LIN {X 0,Y 354.946,Z 276.159,A -85,B 0,C 180,E1 -13383.544,E2 -13383.544} C_VEL
LIN {X 0,Y 356.638,Z 285.927,A -85,B 0,C 180,E1 -13386.173,E2 -13386.173} C_VEL
LIN {X 0,Y 356.254,Z 293.138,A -85,B 0,C 180,E1 -13388.006,E2 -13388.006} C_VEL
LIN {X 0,Y 355.986,Z 296.986,A -85,B 0,C 180,E1 -13388.957,E2 -13388.957} C_VEL
LIN {X 0,Y 356.736,Z 302.12,A -85,B 0,C 180,E1 -13389.429,E2 -13389.429} C_VEL
LIN {X 0,Y 360.066,Z 319.74,A -85,B 0,C 180,E1 -13390.451,E2 -13390.451} C_VEL
LIN {X 0,Y 362.277,Z 335.573,A -85,B 0,C 180,E1 -13391.255,E2 -13391.255} C_VEL
LIN {X 0,Y 363.012,Z 348.096,A -85,B 0,C 180,E1 -13391.771,E2 -13391.771} C_VEL
LIN {X 0,Y 361.012,Z 393.9,A -85,B 0,C 180,E1 -13393.203,E2 -13393.203} C_VEL
LIN {X 0,Y 360.015,Z 405.423,A -85,B 0,C 180,E1 -13393.775,E2 -13393.775} C_VEL
LIN {X 0,Y 359.199,Z 414.432,A -85,B 0,C 180,E1 -13394.393,E2 -13394.393} C_VEL
LIN {X 0,Y 358.156,Z 424.02,A -85,B 0,C 180,E1 -13395.221,E2 -13395.221} C_VEL
LIN {X 0,Y 357.004,Z 434.131,A -85,B 0,C 180,E1 -13396.335,E2 -13396.335} C_VEL
LIN {X 0,Y 356.117,Z 442.074,A -85,B 0,C 180,E1 -13397.462,E2 -13397.462} C_VEL
LIN {X 0,Y 355.278,Z 448.663,A -85,B 0,C 180,E1 -13398.59,E2 -13398.59} C_VEL
LIN {X 0,Y 354.683,Z 454.155,A -85,B 0,C 180,E1 -13399.727,E2 -13399.727} C_VEL
LIN {X 0,Y 354.069,Z 459.784,A -85,B 0,C 180,E1 -13401.151,E2 -13401.151} C_VEL
LIN {X 0,Y 353.657,Z 464.249,A -85,B 0,C 180,E1 -13402.578,E2 -13402.578} C_VEL
LIN {X 0,Y 353.348,Z 468.245,A -85,B 0,C 180,E1 -13404.292,E2 -13404.292} C_VEL
LIN {X 0,Y 353.341,Z 470.093,A -85,B 0,C 180,E1 -13405.436,E2 -13405.436} C_VEL
LIN {X 0,Y 353.398,Z 473.622,A -85,B 0,C 180,E1 -13408.86,E2 -13408.86} C_VEL
LIN {X 0,Y 353.4,Z 474.172,A -85,B 0,C 180,E1 -13410,E2 -13410} C_VEL
LIN {X 0,Y 353.339,Z 474.254,A -85,B 0,C 180,E1 -13411.139,E2 -13411.139} C_VEL
LIN {X 0,Y 353.26,Z 473.86,A -85,B 0,C 180,E1 -13412.28,E2 -13412.28} C_VEL
LIN {X 0,Y 353.269,Z 472.879,A -85,B 0,C 180,E1 -13413.421,E2 -13413.421} C_VEL
LIN {X 0,Y 353.323,Z 470.523,A -85,B 0,C 180,E1 -13415.135,E2 -13415.135} C_VEL
LIN {X 0,Y 353.535,Z 466.838,A -85,B 0,C 180,E1 -13416.85,E2 -13416.85} C_VEL
LIN {X 0,Y 353.807,Z 463.697,A -85,B 0,C 180,E1 -13417.993,E2 -13417.993} C_VEL
LIN {X 0,Y 354.266,Z 458.711,A -85,B 0,C 180,E1 -13419.419,E2 -13419.419} C_VEL
LIN {X 0,Y 354.963,Z 452.453,A -85,B 0,C 180,E1 -13420.841,E2 -13420.841} C_VEL
LIN {X 0,Y 355.656,Z 446.355,A -85,B 0,C 180,E1 -13421.975,E2 -13421.975} C_VEL
LIN {X 0,Y 356.361,Z 439.978,A -85,B 0,C 180,E1 -13422.963,E2 -13422.963} C_VEL
LIN {X 0,Y 357.248,Z 432.28,A -85,B 0,C 180,E1 -13423.945,E2 -13423.945} C_VEL
LIN {X 0,Y 358.02,Z 424.21,A -85,B 0,C 180,E1 -13424.785,E2 -13424.785} C_VEL
LIN {X 0,Y 358.803,Z 415.85,A -85,B 0,C 180,E1 -13425.478,E2 -13425.478} C_VEL
LIN {X 0,Y 359.423,Z 407.491,A -85,B 0,C 180,E1 -13426.023,E2 -13426.023} C_VEL
LIN {X 0,Y 360.085,Z 398.162,A -85,B 0,C 180,E1 -13426.469,E2 -13426.469} C_VEL
LIN {X 0,Y 360.556,Z 386.884,A -85,B 0,C 180,E1 -13426.821,E2 -13426.821} C_VEL
LIN {X 0,Y 361.133,Z 345.094,A -85,B 0,C 180,E1 -13427.675,E2 -13427.675} C_VEL
LIN {X 0,Y 358.638,Z 327.17,A -85,B 0,C 180,E1 -13428.215,E2 -13428.215} C_VEL
LIN {X 0,Y 355.966,Z 312.815,A -85,B 0,C 180,E1 -13428.71,E2 -13428.71} C_VEL
LIN {X 0,Y 357.346,Z 297.3,A -85,B 0,C 180,E1 -13432.676,E2 -13432.676} C_VEL
LIN {X 0,Y 357.807,Z 292.005,A -85,B 0,C 180,E1 -13434.052,E2 -13434.052} C_VEL
LIN {X 0,Y 356.54,Z 283.93,A -85,B 0,C 180,E1 -13436.328,E2 -13436.328} C_VEL
LIN {X 0,Y 354.88,Z 276.094,A -85,B 0,C 180,E1 -13438.684,E2 -13438.684} C_VEL
LIN {X 0,Y 354.795,Z 276.096,A -85,B 0,C 180,E1 -13442.332,E2 -13442.332} C_VEL
LIN {X 0,Y 354.827,Z 276.09,A -85,B 0,C 180,E1 -13445.697,E2 -13445.697} C_VEL
LIN {X 0,Y 354.808,Z 276.101,A -85,B 0,C 180,E1 -13449.417,E2 -13449.417} C_VEL
LIN {X 0,Y 354.796,Z 276.102,A -85,B 0,C 180,E1 -13452.865,E2 -13452.865} C_VEL
LIN {X 0,Y 354.775,Z 276.104,A -85,B 0,C 180,E1 -13456.102,E2 -13456.102} C_VEL
LIN {X 0,Y 354.774,Z 276.105,A -85,B 0,C 180,E1 -13459.174,E2 -13459.174} C_VEL
LIN {X 0,Y 354.808,Z 276.099,A -85,B 0,C 180,E1 -13462.402,E2 -13462.402} C_VEL
LIN {X 0,Y 354.819,Z 276.092,A -85,B 0,C 180,E1 -13464.939,E2 -13464.939} C_VEL
LIN {X 0,Y 354.8,Z 276.094,A -85,B 0,C 180,E1 -13468.403,E2 -13468.403} C_VEL
LIN {X 0,Y 354.81,Z 276.103,A -85,B 0,C 180,E1 -13471.612,E2 -13471.612} C_VEL
LIN {X 0,Y 354.858,Z 276.093,A -85,B 0,C 180,E1 -13475.421,E2 -13475.421} C_VEL
LIN {X 0,Y 354.833,Z 276.087,A -85,B 0,C 180,E1 -13479.11,E2 -13479.11} C_VEL
LIN {X 0,Y 354.885,Z 276.084,A -85,B 0,C 180,E1 -13482.716,E2 -13482.716} C_VEL
LIN {X 0,Y 354.956,Z 276.08,A -85,B 0,C 180,E1 -13486.252,E2 -13486.252} C_VEL
LIN {X 0,Y 354.981,Z 276.068,A -85,B 0,C 180,E1 -13489.733,E2 -13489.733} C_VEL
LIN {X 0,Y 355.127,Z 276.053,A -85,B 0,C 180,E1 -13493.177,E2 -13493.177} C_VEL
LIN {X 0,Y 355.234,Z 276.044,A -85,B 0,C 180,E1 -13497.729,E2 -13497.729} C_VEL
LIN {X 0,Y 355.352,Z 276.022,A -85,B 0,C 180,E1 -13499.996,E2 -13499.996} C_VEL
LIN {X 0,Y 355.24,Z 276.047,A -85,B 0,C 180,E1 -13502.264,E2 -13502.264} C_VEL
LIN {X 0,Y 355.096,Z 276.061,A -85,B 0,C 180,E1 -13506.816,E2 -13506.816} C_VEL
LIN {X 0,Y 354.951,Z 276.076,A -85,B 0,C 180,E1 -13510.261,E2 -13510.261} C_VEL
LIN {X 0,Y 354.937,Z 276.086,A -85,B 0,C 180,E1 -13514.015,E2 -13514.015} C_VEL
LIN {X 0,Y 354.914,Z 276.088,A -85,B 0,C 180,E1 -13518.104,E2 -13518.104} C_VEL
LIN {X 0,Y 354.824,Z 276.098,A -85,B 0,C 180,E1 -13522.102,E2 -13522.102} C_VEL
LIN {X 0,Y 354.887,Z 276.088,A -85,B 0,C 180,E1 -13525.823,E2 -13525.823} C_VEL
LIN {X 0,Y 354.803,Z 276.1,A -85,B 0,C 180,E1 -13529.678,E2 -13529.678} C_VEL
LIN {X 0,Y 354.789,Z 276.102,A -85,B 0,C 180,E1 -13533.698,E2 -13533.698} C_VEL
LIN {X 0,Y 354.779,Z 276.093,A -85,B 0,C 180,E1 -13536.456,E2 -13536.456} C_VEL
LIN {X 0,Y 354.804,Z 276.097,A -85,B 0,C 180,E1 -13539.42,E2 -13539.42} C_VEL
LIN {X 0,Y 354.819,Z 276.1,A -85,B 0,C 180,E1 -13542.873,E2 -13542.873} C_VEL
LIN {X 0,Y 354.844,Z 276.098,A -85,B 0,C 180,E1 -13546.116,E2 -13546.116} C_VEL
LIN {X 0,Y 354.831,Z 276.097,A -85,B 0,C 180,E1 -13549.185,E2 -13549.185} C_VEL
LIN {X 0,Y 354.844,Z 276.163,A -85,B 0,C 180,E1 -13552.213,E2 -13552.213} C_VEL
LIN {X 0,Y 356.19,Z 282.921,A -85,B 0,C 180,E1 -13554.336,E2 -13554.336} C_VEL
LIN {X 0,Y 359.045,Z 291.373,A -85,B 0,C 180,E1 -13554.722,E2 -13554.722} C_VEL
LIN {X 0,Y 361.86,Z 303.963,A -85,B 0,C 180,E1 -13555.175,E2 -13555.175} C_VEL
LIN {X 0,Y 360.834,Z 359.468,A -85,B 0,C 180,E1 -13556.325,E2 -13556.325} C_VEL
LIN {X 0,Y 360.551,Z 369.013,A -85,B 0,C 180,E1 -13556.672,E2 -13556.672} C_VEL
LIN {X 0,Y 360.038,Z 379.383,A -85,B 0,C 180,E1 -13557.226,E2 -13557.226} C_VEL
LIN {X 0,Y 359.213,Z 390.94,A -85,B 0,C 180,E1 -13558.113,E2 -13558.113} C_VEL
LIN {X 0,Y 358.442,Z 399.876,A -85,B 0,C 180,E1 -13559.024,E2 -13559.024} C_VEL
LIN {X 0,Y 357.714,Z 407.018,A -85,B 0,C 180,E1 -13559.919,E2 -13559.919} C_VEL
LIN {X 0,Y 356.986,Z 413.17,A -85,B 0,C 180,E1 -13560.84,E2 -13560.84} C_VEL
LIN {X 0,Y 356.21,Z 419.701,A -85,B 0,C 180,E1 -13562.025,E2 -13562.025} C_VEL
LIN {X 0,Y 355.528,Z 425.327,A -85,B 0,C 180,E1 -13563.275,E2 -13563.275} C_VEL
LIN {X 0,Y 354.957,Z 429.812,A -85,B 0,C 180,E1 -13564.492,E2 -13564.492} C_VEL
LIN {X 0,Y 354.325,Z 434.751,A -85,B 0,C 180,E1 -13566.199,E2 -13566.199} C_VEL
LIN {X 0,Y 353.87,Z 438.18,A -85,B 0,C 180,E1 -13567.831,E2 -13567.831} C_VEL
LIN {X 0,Y 353.582,Z 439.976,A -85,B 0,C 180,E1 -13569.083,E2 -13569.083} C_VEL
LIN {X 0,Y 353.408,Z 441.07,A -85,B 0,C 180,E1 -13570.241,E2 -13570.241} C_VEL
LIN {X 0,Y 353.252,Z 441.693,A -85,B 0,C 180,E1 -13571.439,E2 -13571.439} C_VEL
LIN {X 0,Y 353.202,Z 441.763,A -85,B 0,C 180,E1 -13572.747,E2 -13572.747} C_VEL
LIN {X 0,Y 353.22,Z 441.38,A -85,B 0,C 180,E1 -13573.826,E2 -13573.826} C_VEL
LIN {X 0,Y 353.277,Z 440.368,A -85,B 0,C 180,E1 -13575.012,E2 -13575.012} C_VEL
LIN {X 0,Y 353.478,Z 437.505,A -85,B 0,C 180,E1 -13576.941,E2 -13576.941} C_VEL
LIN {X 0,Y 353.723,Z 433.912,A -85,B 0,C 180,E1 -13578.54,E2 -13578.54} C_VEL
LIN {X 0,Y 354.107,Z 428.587,A -85,B 0,C 180,E1 -13580.288,E2 -13580.288} C_VEL
LIN {X 0,Y 354.55,Z 421.521,A -85,B 0,C 180,E1 -13582.024,E2 -13582.024} C_VEL
LIN {X 0,Y 355.033,Z 415.532,A -85,B 0,C 180,E1 -13583.179,E2 -13583.179} C_VEL
LIN {X 0,Y 355.565,Z 408.244,A -85,B 0,C 180,E1 -13584.328,E2 -13584.328} C_VEL
LIN {X 0,Y 356.102,Z 400.466,A -85,B 0,C 180,E1 -13585.331,E2 -13585.331} C_VEL
LIN {X 0,Y 356.605,Z 392.284,A -85,B 0,C 180,E1 -13586.186,E2 -13586.186} C_VEL
LIN {X 0,Y 357.064,Z 383.771,A -85,B 0,C 180,E1 -13586.897,E2 -13586.897} C_VEL
LIN {X 0,Y 357.499,Z 373.816,A -85,B 0,C 180,E1 -13587.536,E2 -13587.536} C_VEL
LIN {X 0,Y 357.829,Z 361.516,A -85,B 0,C 180,E1 -13588.066,E2 -13588.066} C_VEL
LIN {X 0,Y 358.085,Z 341.16,A -85,B 0,C 180,E1 -13588.524,E2 -13588.524} C_VEL
LIN {X 0,Y 358.615,Z 301.683,A -85,B 0,C 180,E1 -13589.313,E2 -13589.313} C_VEL
LIN {X 0,Y 355.434,Z 282.466,A -85,B 0,C 180,E1 -13589.856,E2 -13589.856} C_VEL
LIN {X 0,Y 355.45,Z 278.059,A -85,B 0,C 180,E1 -13591.133,E2 -13591.133} C_VEL
LIN {X 0,Y 355.224,Z 276.047,A -85,B 0,C 180,E1 -13591.772,E2 -13591.772} C_VEL
LIN {X 0,Y 355.091,Z 276.065,A -85,B 0,C 180,E1 -13596.82,E2 -13596.82} C_VEL
LIN {X 0,Y 354.943,Z 276.081,A -85,B 0,C 180,E1 -13600.265,E2 -13600.265} C_VEL
LIN {X 0,Y 354.909,Z 276.085,A -85,B 0,C 180,E1 -13604.02,E2 -13604.02} C_VEL
LIN {X 0,Y 354.89,Z 276.087,A -85,B 0,C 180,E1 -13608.11,E2 -13608.11} C_VEL
LIN {X 0,Y 354.798,Z 276.099,A -85,B 0,C 180,E1 -13612.109,E2 -13612.109} C_VEL
LIN {X 0,Y 354.781,Z 276.103,A -85,B 0,C 180,E1 -13613.617,E2 -13613.617} C_VEL
LIN {X 0,Y 354.105,Z 276.186,A -85,B 0,C 180,E1 -13614.565,E2 -13614.565} C_VEL
LIN {X 0,Y 351.218,Z 276.545,A -85,B 0,C 180,E1 -13616.106,E2 -13616.106} C_VEL
LIN {X 0,Y 348.787,Z 276.853,A -85,B 0,C 180,E1 -13617.352,E2 -13617.352} C_VEL
LIN {X 0,Y 347.766,Z 276.975,A -85,B 0,C 180,E1 -13618.318,E2 -13618.318} C_VEL
LIN {X 0,Y 347.695,Z 276.983,A -85,B 0,C 180,E1 -13618.645,E2 -13618.645} C_VEL
LIN {X 0,Y 347.71,Z 276.984,A -85,B 0,C 180,E1 -13621.917,E2 -13621.917} C_VEL
LIN {X 0,Y 347.761,Z 276.979,A -85,B 0,C 180,E1 -13625.879,E2 -13625.879} C_VEL
LIN {X 0,Y 347.706,Z 276.982,A -85,B 0,C 180,E1 -13628.799,E2 -13628.799} C_VEL
LIN {X 0,Y 347.72,Z 276.985,A -85,B 0,C 180,E1 -13631.835,E2 -13631.835} C_VEL
LIN {X 0,Y 347.683,Z 276.986,A -85,B 0,C 180,E1 -13635.031,E2 -13635.031} C_VEL
LIN {X 0,Y 347.731,Z 276.98,A -85,B 0,C 180,E1 -13638.401,E2 -13638.401} C_VEL
LIN {X 0,Y 347.755,Z 276.98,A -85,B 0,C 180,E1 -13642.016,E2 -13642.016} C_VEL
LIN {X 0,Y 347.729,Z 276.982,A -85,B 0,C 180,E1 -13645.54,E2 -13645.54} C_VEL
LIN {X 0,Y 347.731,Z 276.982,A -85,B 0,C 180,E1 -13648.305,E2 -13648.305} C_VEL
LIN {X 0,Y 347.733,Z 276.979,A -85,B 0,C 180,E1 -13650.989,E2 -13650.989} C_VEL
LIN {X 0,Y 347.74,Z 276.981,A -85,B 0,C 180,E1 -13653.605,E2 -13653.605} C_VEL
LIN {X 0,Y 347.76,Z 276.98,A -85,B 0,C 180,E1 -13656.165,E2 -13656.165} C_VEL
LIN {X 0,Y 347.806,Z 276.975,A -85,B 0,C 180,E1 -13659.914,E2 -13659.914} C_VEL
LIN {X 0,Y 347.971,Z 277.138,A -85,B 0,C 180,E1 -13662.597,E2 -13662.597} C_VEL
LIN {X 0,Y 347.912,Z 281.643,A -85,B 0,C 180,E1 -13663.795,E2 -13663.795} C_VEL
LIN {X 0,Y 350.542,Z 302.01,A -85,B 0,C 180,E1 -13664.442,E2 -13664.442} C_VEL
LIN {X 0,Y 349.342,Z 360.728,A -85,B 0,C 180,E1 -13666.109,E2 -13666.109} C_VEL
LIN {X 0,Y 349.119,Z 370.424,A -85,B 0,C 180,E1 -13666.545,E2 -13666.545} C_VEL
LIN {X 0,Y 348.777,Z 380.963,A -85,B 0,C 180,E1 -13667.198,E2 -13667.198} C_VEL
LIN {X 0,Y 348.416,Z 391.533,A -85,B 0,C 180,E1 -13668.072,E2 -13668.072} C_VEL
LIN {X 0,Y 347.964,Z 400.972,A -85,B 0,C 180,E1 -13669.089,E2 -13669.089} C_VEL
LIN {X 0,Y 347.487,Z 409.704,A -85,B 0,C 180,E1 -13670.252,E2 -13670.252} C_VEL
LIN {X 0,Y 347.094,Z 417.664,A -85,B 0,C 180,E1 -13671.563,E2 -13671.563} C_VEL
LIN {X 0,Y 346.798,Z 424.606,A -85,B 0,C 180,E1 -13673.02,E2 -13673.02} C_VEL
LIN {X 0,Y 346.581,Z 429.149,A -85,B 0,C 180,E1 -13674.185,E2 -13674.185} C_VEL
LIN {X 0,Y 346.445,Z 434.513,A -85,B 0,C 180,E1 -13675.932,E2 -13675.932} C_VEL
LIN {X 0,Y 346.25,Z 438.421,A -85,B 0,C 180,E1 -13677.677,E2 -13677.677} C_VEL
LIN {X 0,Y 346.239,Z 440.213,A -85,B 0,C 180,E1 -13678.841,E2 -13678.841} C_VEL
LIN {X 0,Y 346.27,Z 441.417,A -85,B 0,C 180,E1 -13680.004,E2 -13680.004} C_VEL
LIN {X 0,Y 346.341,Z 442.092,A -85,B 0,C 180,E1 -13681.166,E2 -13681.166} C_VEL
LIN {X 0,Y 346.501,Z 442.245,A -85,B 0,C 180,E1 -13682.329,E2 -13682.329} C_VEL
LIN {X 0,Y 346.775,Z 441.869,A -85,B 0,C 180,E1 -13683.489,E2 -13683.489} C_VEL
LIN {X 0,Y 347.098,Z 440.938,A -85,B 0,C 180,E1 -13684.649,E2 -13684.649} C_VEL
LIN {X 0,Y 347.375,Z 438.425,A -85,B 0,C 180,E1 -13686.392,E2 -13686.392} C_VEL
LIN {X 0,Y 347.721,Z 436.096,A -85,B 0,C 180,E1 -13687.553,E2 -13687.553} C_VEL
LIN {X 0,Y 348.335,Z 433.25,A -85,B 0,C 180,E1 -13688.648,E2 -13688.648} C_VEL
LIN {X 0,Y 349.063,Z 428.307,A -85,B 0,C 180,E1 -13690.15,E2 -13690.15} C_VEL
LIN {X 0,Y 349.983,Z 422.239,A -85,B 0,C 180,E1 -13691.588,E2 -13691.588} C_VEL
LIN {X 0,Y 350.929,Z 416.282,A -85,B 0,C 180,E1 -13692.73,E2 -13692.73} C_VEL
LIN {X 0,Y 351.89,Z 409.106,A -85,B 0,C 180,E1 -13693.87,E2 -13693.87} C_VEL
LIN {X 0,Y 353.105,Z 399.17,A -85,B 0,C 180,E1 -13695.146,E2 -13695.146} C_VEL
LIN {X 0,Y 354.14,Z 389.136,A -85,B 0,C 180,E1 -13696.134,E2 -13696.134} C_VEL
LIN {X 0,Y 355.129,Z 378.103,A -85,B 0,C 180,E1 -13696.975,E2 -13696.975} C_VEL
LIN {X 0,Y 355.836,Z 367.087,A -85,B 0,C 180,E1 -13697.57,E2 -13697.57} C_VEL
LIN {X 0,Y 356.406,Z 355.874,A -85,B 0,C 180,E1 -13697.986,E2 -13697.986} C_VEL
LIN {X 0,Y 358.797,Z 307.744,A -85,B 0,C 180,E1 -13699.509,E2 -13699.509} C_VEL
LIN {X 0,Y 356.388,Z 298.357,A -85,B 0,C 180,E1 -13700.132,E2 -13700.132} C_VEL
LIN {X 0,Y 351.659,Z 288.448,A -85,B 0,C 180,E1 -13701.087,E2 -13701.087} C_VEL
LIN {X 0,Y 350.011,Z 285.153,A -85,B 0,C 180,E1 -13701.448,E2 -13701.448} C_VEL
LIN {X 0,Y 347.793,Z 276.978,A -85,B 0,C 180,E1 -13704.291,E2 -13704.291} C_VEL
LIN {X 0,Y 347.747,Z 276.981,A -85,B 0,C 180,E1 -13707.702,E2 -13707.702} C_VEL
LIN {X 0,Y 347.748,Z 276.983,A -85,B 0,C 180,E1 -13710.351,E2 -13710.351} C_VEL
LIN {X 0,Y 347.758,Z 276.98,A -85,B 0,C 180,E1 -13714.046,E2 -13714.046} C_VEL
LIN {X 0,Y 347.765,Z 276.979,A -85,B 0,C 180,E1 -13717.323,E2 -13717.323} C_VEL
LIN {X 0,Y 347.751,Z 276.979,A -85,B 0,C 180,E1 -13721.602,E2 -13721.602} C_VEL
LIN {X 0,Y 347.715,Z 276.983,A -85,B 0,C 180,E1 -13725.028,E2 -13725.028} C_VEL
LIN {X 0,Y 347.759,Z 276.979,A -85,B 0,C 180,E1 -13728.399,E2 -13728.399} C_VEL
LIN {X 0,Y 347.773,Z 276.977,A -85,B 0,C 180,E1 -13732.015,E2 -13732.015} C_VEL
LIN {X 0,Y 347.754,Z 276.977,A -85,B 0,C 180,E1 -13735.537,E2 -13735.537} C_VEL
LIN {X 0,Y 347.754,Z 276.976,A -85,B 0,C 180,E1 -13738.301,E2 -13738.301} C_VEL
LIN {X 0,Y 347.788,Z 276.973,A -85,B 0,C 180,E1 -13740.988,E2 -13740.988} C_VEL
LIN {X 0,Y 347.947,Z 277.152,A -85,B 0,C 180,E1 -13743.417,E2 -13743.417} C_VEL
LIN {X 0,Y 349.677,Z 287.663,A -85,B 0,C 180,E1 -13746.298,E2 -13746.298} C_VEL
LIN {X 0,Y 349.249,Z 293.864,A -85,B 0,C 180,E1 -13747.861,E2 -13747.861} C_VEL
LIN {X 0,Y 350.304,Z 301.781,A -85,B 0,C 180,E1 -13748.668,E2 -13748.668} C_VEL
LIN {X 0,Y 352.854,Z 314.237,A -85,B 0,C 180,E1 -13749.469,E2 -13749.469} C_VEL
LIN {X 0,Y 355.698,Z 332.426,A -85,B 0,C 180,E1 -13750.493,E2 -13750.493} C_VEL
LIN {X 0,Y 356.803,Z 345.41,A -85,B 0,C 180,E1 -13751.091,E2 -13751.091} C_VEL
LIN {X 0,Y 356.545,Z 355.218,A -85,B 0,C 180,E1 -13751.432,E2 -13751.432} C_VEL
LIN {X 0,Y 354.694,Z 393.678,A -85,B 0,C 180,E1 -13752.682,E2 -13752.682} C_VEL
LIN {X 0,Y 353.535,Z 406.057,A -85,B 0,C 180,E1 -13753.321,E2 -13753.321} C_VEL
LIN {X 0,Y 352.69,Z 414.859,A -85,B 0,C 180,E1 -13753.949,E2 -13753.949} C_VEL
LIN {X 0,Y 351.569,Z 424.242,A -85,B 0,C 180,E1 -13754.789,E2 -13754.789} C_VEL
LIN {X 0,Y 350.302,Z 434.112,A -85,B 0,C 180,E1 -13755.921,E2 -13755.921} C_VEL
LIN {X 0,Y 349.256,Z 442.827,A -85,B 0,C 180,E1 -13757.211,E2 -13757.211} C_VEL
LIN {X 0,Y 348.349,Z 449.252,A -85,B 0,C 180,E1 -13758.36,E2 -13758.36} C_VEL
LIN {X 0,Y 347.577,Z 455.836,A -85,B 0,C 180,E1 -13759.809,E2 -13759.809} C_VEL
LIN {X 0,Y 346.952,Z 461.074,A -85,B 0,C 180,E1 -13761.261,E2 -13761.261} C_VEL
LIN {X 0,Y 346.459,Z 465.764,A -85,B 0,C 180,E1 -13763.009,E2 -13763.009} C_VEL
LIN {X 0,Y 346.278,Z 468.171,A -85,B 0,C 180,E1 -13764.175,E2 -13764.175} C_VEL
LIN {X 0,Y 346.253,Z 469.983,A -85,B 0,C 180,E1 -13765.343,E2 -13765.343} C_VEL
LIN {X 0,Y 346.302,Z 473.234,A -85,B 0,C 180,E1 -13768.837,E2 -13768.837} C_VEL
LIN {X 0,Y 346.321,Z 473.825,A -85,B 0,C 180,E1 -13770,E2 -13770} C_VEL
LIN {X 0,Y 346.242,Z 473.945,A -85,B 0,C 180,E1 -13771.163,E2 -13771.163} C_VEL
LIN {X 0,Y 346.166,Z 473.572,A -85,B 0,C 180,E1 -13772.327,E2 -13772.327} C_VEL
LIN {X 0,Y 346.192,Z 472.609,A -85,B 0,C 180,E1 -13773.491,E2 -13773.491} C_VEL
LIN {X 0,Y 346.249,Z 471.15,A -85,B 0,C 180,E1 -13774.657,E2 -13774.657} C_VEL
LIN {X 0,Y 346.359,Z 468.023,A -85,B 0,C 180,E1 -13776.407,E2 -13776.407} C_VEL
LIN {X 0,Y 346.765,Z 463.594,A -85,B 0,C 180,E1 -13778.156,E2 -13778.156} C_VEL
LIN {X 0,Y 347.413,Z 457.506,A -85,B 0,C 180,E1 -13779.901,E2 -13779.901} C_VEL
LIN {X 0,Y 347.985,Z 452.497,A -85,B 0,C 180,E1 -13781.061,E2 -13781.061} C_VEL
LIN {X 0,Y 348.711,Z 446.481,A -85,B 0,C 180,E1 -13782.217,E2 -13782.217} C_VEL
LIN {X 0,Y 349.597,Z 439.179,A -85,B 0,C 180,E1 -13783.367,E2 -13783.367} C_VEL
LIN {X 0,Y 350.384,Z 432.614,A -85,B 0,C 180,E1 -13784.224,E2 -13784.224} C_VEL
LIN {X 0,Y 351.192,Z 424.688,A -85,B 0,C 180,E1 -13785.079,E2 -13785.079} C_VEL
LIN {X 0,Y 352.002,Z 416.528,A -85,B 0,C 180,E1 -13785.785,E2 -13785.785} C_VEL
LIN {X 0,Y 352.658,Z 408.368,A -85,B 0,C 180,E1 -13786.345,E2 -13786.345} C_VEL
LIN {X 0,Y 353.316,Z 399.843,A -85,B 0,C 180,E1 -13786.783,E2 -13786.783} C_VEL
LIN {X 0,Y 353.753,Z 390.385,A -85,B 0,C 180,E1 -13787.123,E2 -13787.123} C_VEL
LIN {X 0,Y 354.417,Z 344.786,A -85,B 0,C 180,E1 -13788.104,E2 -13788.104} C_VEL
LIN {X 0,Y 351.62,Z 325.662,A -85,B 0,C 180,E1 -13788.705,E2 -13788.705} C_VEL
LIN {X 0,Y 349.106,Z 312.402,A -85,B 0,C 180,E1 -13789.194,E2 -13789.194} C_VEL
LIN {X 0,Y 350.673,Z 296.559,A -85,B 0,C 180,E1 -13793.336,E2 -13793.336} C_VEL
LIN {X 0,Y 350.874,Z 293.168,A -85,B 0,C 180,E1 -13794.243,E2 -13794.243} C_VEL
LIN {X 0,Y 349.557,Z 285.101,A -85,B 0,C 180,E1 -13796.573,E2 -13796.573} C_VEL
LIN {X 0,Y 347.825,Z 276.971,A -85,B 0,C 180,E1 -13799.064,E2 -13799.064} C_VEL
LIN {X 0,Y 347.742,Z 276.977,A -85,B 0,C 180,E1 -13803.071,E2 -13803.071} C_VEL
LIN {X 0,Y 347.775,Z 276.968,A -85,B 0,C 180,E1 -13806.063,E2 -13806.063} C_VEL
LIN {X 0,Y 347.739,Z 276.981,A -85,B 0,C 180,E1 -13808.794,E2 -13808.794} C_VEL
LIN {X 0,Y 347.758,Z 276.978,A -85,B 0,C 180,E1 -13811.829,E2 -13811.829} C_VEL
LIN {X 0,Y 347.713,Z 276.981,A -85,B 0,C 180,E1 -13815.025,E2 -13815.025} C_VEL
LIN {X 0,Y 347.75,Z 276.978,A -85,B 0,C 180,E1 -13818.397,E2 -13818.397} C_VEL
LIN {X 0,Y 347.764,Z 276.976,A -85,B 0,C 180,E1 -13822.676,E2 -13822.676} C_VEL
LIN {X 0,Y 347.756,Z 276.979,A -85,B 0,C 180,E1 -13825.954,E2 -13825.954} C_VEL
LIN {X 0,Y 347.746,Z 276.975,A -85,B 0,C 180,E1 -13829.649,E2 -13829.649} C_VEL
LIN {X 0,Y 347.765,Z 276.972,A -85,B 0,C 180,E1 -13833.599,E2 -13833.599} C_VEL
LIN {X 0,Y 347.78,Z 276.976,A -85,B 0,C 180,E1 -13836.158,E2 -13836.158} C_VEL
LIN {X 0,Y 347.806,Z 276.97,A -85,B 0,C 180,E1 -13839.906,E2 -13839.906} C_VEL
LIN {X 0,Y 347.837,Z 276.96,A -85,B 0,C 180,E1 -13843.565,E2 -13843.565} C_VEL
LIN {X 0,Y 347.894,Z 276.957,A -85,B 0,C 180,E1 -13847.157,E2 -13847.157} C_VEL
LIN {X 0,Y 347.948,Z 276.949,A -85,B 0,C 180,E1 -13850.698,E2 -13850.698} C_VEL
LIN {X 0,Y 348.093,Z 276.929,A -85,B 0,C 180,E1 -13853.039,E2 -13853.039} C_VEL
LIN {X 0,Y 348.196,Z 276.921,A -85,B 0,C 180,E1 -13857.683,E2 -13857.683} C_VEL
LIN {X 0,Y 348.303,Z 276.9,A -85,B 0,C 180,E1 -13859.996,E2 -13859.996} C_VEL
LIN {X 0,Y 348.202,Z 276.923,A -85,B 0,C 180,E1 -13862.31,E2 -13862.31} C_VEL
LIN {X 0,Y 348.064,Z 276.937,A -85,B 0,C 180,E1 -13866.954,E2 -13866.954} C_VEL
LIN {X 0,Y 347.892,Z 276.954,A -85,B 0,C 180,E1 -13870.471,E2 -13870.471} C_VEL
LIN {X 0,Y 347.892,Z 276.963,A -85,B 0,C 180,E1 -13874.146,E2 -13874.146} C_VEL
LIN {X 0,Y 347.882,Z 276.966,A -85,B 0,C 180,E1 -13878.286,E2 -13878.286} C_VEL
LIN {X 0,Y 347.779,Z 276.972,A -85,B 0,C 180,E1 -13881.631,E2 -13881.631} C_VEL
LIN {X 0,Y 347.8,Z 276.97,A -85,B 0,C 180,E1 -13885.104,E2 -13885.104} C_VEL
LIN {X 0,Y 347.794,Z 276.972,A -85,B 0,C 180,E1 -13887.69,E2 -13887.69} C_VEL
LIN {X 0,Y 347.734,Z 276.985,A -85,B 0,C 180,E1 -13890.344,E2 -13890.344} C_VEL
LIN {X 0,Y 347.731,Z 276.983,A -85,B 0,C 180,E1 -13894.04,E2 -13894.04} C_VEL
LIN {X 0,Y 347.742,Z 276.98,A -85,B 0,C 180,E1 -13897.317,E2 -13897.317} C_VEL
LIN {X 0,Y 347.773,Z 276.97,A -85,B 0,C 180,E1 -13900.285,E2 -13900.285} C_VEL
LIN {X 0,Y 347.797,Z 276.971,A -85,B 0,C 180,E1 -13903.39,E2 -13903.39} C_VEL
LIN {X 0,Y 347.794,Z 276.972,A -85,B 0,C 180,E1 -13906.667,E2 -13906.667} C_VEL
LIN {X 0,Y 347.76,Z 276.981,A -85,B 0,C 180,E1 -13910.162,E2 -13910.162} C_VEL
LIN {X 0,Y 347.817,Z 277.184,A -85,B 0,C 180,E1 -13911.881,E2 -13911.881} C_VEL
LIN {X 0,Y 349.092,Z 283.487,A -85,B 0,C 180,E1 -13913.862,E2 -13913.862} C_VEL
LIN {X 0,Y 352.613,Z 293.121,A -85,B 0,C 180,E1 -13914.326,E2 -13914.326} C_VEL
LIN {X 0,Y 355.249,Z 304.815,A -85,B 0,C 180,E1 -13914.761,E2 -13914.761} C_VEL
LIN {X 0,Y 354.224,Z 359.623,A -85,B 0,C 180,E1 -13915.919,E2 -13915.919} C_VEL
LIN {X 0,Y 353.916,Z 368.874,A -85,B 0,C 180,E1 -13916.255,E2 -13916.255} C_VEL
LIN {X 0,Y 353.441,Z 379.002,A -85,B 0,C 180,E1 -13916.8,E2 -13916.8} C_VEL
LIN {X 0,Y 352.606,Z 389.917,A -85,B 0,C 180,E1 -13917.611,E2 -13917.611} C_VEL
LIN {X 0,Y 351.807,Z 399.111,A -85,B 0,C 180,E1 -13918.541,E2 -13918.541} C_VEL
LIN {X 0,Y 350.971,Z 407.008,A -85,B 0,C 180,E1 -13919.533,E2 -13919.533} C_VEL
LIN {X 0,Y 350.156,Z 413.651,A -85,B 0,C 180,E1 -13920.545,E2 -13920.545} C_VEL
LIN {X 0,Y 349.486,Z 418.802,A -85,B 0,C 180,E1 -13921.472,E2 -13921.472} C_VEL
LIN {X 0,Y 348.777,Z 424.518,A -85,B 0,C 180,E1 -13922.715,E2 -13922.715} C_VEL
LIN {X 0,Y 348.151,Z 429.218,A -85,B 0,C 180,E1 -13923.956,E2 -13923.956} C_VEL
LIN {X 0,Y 347.489,Z 433.869,A -85,B 0,C 180,E1 -13925.51,E2 -13925.51} C_VEL
LIN {X 0,Y 347.08,Z 436.762,A -85,B 0,C 180,E1 -13926.743,E2 -13926.743} C_VEL
LIN {X 0,Y 346.551,Z 440.232,A -85,B 0,C 180,E1 -13928.871,E2 -13928.871} C_VEL
LIN {X 0,Y 346.2,Z 441.95,A -85,B 0,C 180,E1 -13931.046,E2 -13931.046} C_VEL
LIN {X 0,Y 346.121,Z 442.111,A -85,B 0,C 180,E1 -13932.599,E2 -13932.599} C_VEL
LIN {X 0,Y 346.11,Z 441.853,A -85,B 0,C 180,E1 -13933.484,E2 -13933.484} C_VEL
LIN {X 0,Y 346.153,Z 440.935,A -85,B 0,C 180,E1 -13934.696,E2 -13934.696} C_VEL
LIN {X 0,Y 346.382,Z 438.012,A -85,B 0,C 180,E1 -13936.857,E2 -13936.857} C_VEL
LIN {X 0,Y 346.604,Z 434.965,A -85,B 0,C 180,E1 -13938.301,E2 -13938.301} C_VEL
LIN {X 0,Y 346.809,Z 431.78,A -85,B 0,C 180,E1 -13939.492,E2 -13939.492} C_VEL
LIN {X 0,Y 347.211,Z 426.689,A -85,B 0,C 180,E1 -13940.975,E2 -13940.975} C_VEL
LIN {X 0,Y 347.638,Z 420.583,A -85,B 0,C 180,E1 -13942.39,E2 -13942.39} C_VEL
LIN {X 0,Y 348.149,Z 413.998,A -85,B 0,C 180,E1 -13943.626,E2 -13943.626} C_VEL
LIN {X 0,Y 348.595,Z 407.394,A -85,B 0,C 180,E1 -13944.65,E2 -13944.65} C_VEL
LIN {X 0,Y 349.209,Z 399.357,A -85,B 0,C 180,E1 -13945.672,E2 -13945.672} C_VEL
LIN {X 0,Y 349.846,Z 389.325,A -85,B 0,C 180,E1 -13946.689,E2 -13946.689} C_VEL
LIN {X 0,Y 350.347,Z 378.642,A -85,B 0,C 180,E1 -13947.485,E2 -13947.485} C_VEL
LIN {X 0,Y 350.714,Z 368.547,A -85,B 0,C 180,E1 -13948.026,E2 -13948.026} C_VEL
LIN {X 0,Y 350.905,Z 359.785,A -85,B 0,C 180,E1 -13948.35,E2 -13948.35} C_VEL
LIN {X 0,Y 351.703,Z 302.619,A -85,B 0,C 180,E1 -13949.55,E2 -13949.55} C_VEL
LIN {X 0,Y 348.471,Z 282.817,A -85,B 0,C 180,E1 -13950.109,E2 -13950.109} C_VEL
LIN {X 0,Y 348.228,Z 277.116,A -85,B 0,C 180,E1 -13951.807,E2 -13951.807} C_VEL
LIN {X 0,Y 348.057,Z 276.942,A -85,B 0,C 180,E1 -13956.959,E2 -13956.959} C_VEL
LIN {X 0,Y 347.894,Z 276.959,A -85,B 0,C 180,E1 -13960.476,E2 -13960.476} C_VEL
LIN {X 0,Y 347.866,Z 276.962,A -85,B 0,C 180,E1 -13964.151,E2 -13964.151} C_VEL
LIN {X 0,Y 347.858,Z 276.963,A -85,B 0,C 180,E1 -13968.292,E2 -13968.292} C_VEL
LIN {X 0,Y 347.755,Z 276.98,A -85,B 0,C 180,E1 -13971.636,E2 -13971.636} C_VEL
LIN {X 0,Y 347.739,Z 276.981,A -85,B 0,C 180,E1 -13975.114,E2 -13975.114} C_VEL
LIN {X 0,Y 347.695,Z 276.983,A -85,B 0,C 180,E1 -13978.645,E2 -13978.645} C_VEL
LIN {X 0,Y 347.047,Z 277.069,A -85,B 0,C 180,E1 -13979.612,E2 -13979.612} C_VEL
LIN {X 0,Y 344.163,Z 277.426,A -85,B 0,C 180,E1 -13981.183,E2 -13981.183} C_VEL
LIN {X 0,Y 341.73,Z 277.727,A -85,B 0,C 180,E1 -13982.456,E2 -13982.456} C_VEL
LIN {X 0,Y 340.722,Z 277.857,A -85,B 0,C 180,E1 -13983.442,E2 -13983.442} C_VEL
LIN {X 0,Y 340.66,Z 277.862,A -85,B 0,C 180,E1 -13983.776,E2 -13983.776} C_VEL
LIN {X 0,Y 340.676,Z 277.858,A -85,B 0,C 180,E1 -13986.746,E2 -13986.746} C_VEL
LIN {X 0,Y 340.627,Z 277.865,A -85,B 0,C 180,E1 -13990.243,E2 -13990.243} C_VEL
LIN {X 0,Y 340.651,Z 277.861,A -85,B 0,C 180,E1 -13992.909,E2 -13992.909} C_VEL
LIN {X 0,Y 340.656,Z 277.861,A -85,B 0,C 180,E1 -13997.1,E2 -13997.1} C_VEL
LIN {X 0,Y 340.681,Z 277.859,A -85,B 0,C 180,E1 -14000.252,E2 -14000.252} C_VEL
LIN {X 0,Y 340.693,Z 277.859,A -85,B 0,C 180,E1 -14003.564,E2 -14003.564} C_VEL
LIN {X 0,Y 340.677,Z 277.861,A -85,B 0,C 180,E1 -14006.158,E2 -14006.158} C_VEL
LIN {X 0,Y 340.708,Z 277.859,A -85,B 0,C 180,E1 -14010.039,E2 -14010.039} C_VEL
LIN {X 0,Y 340.71,Z 277.854,A -85,B 0,C 180,E1 -14013.017,E2 -14013.017} C_VEL
LIN {X 0,Y 340.732,Z 277.854,A -85,B 0,C 180,E1 -14015.642,E2 -14015.642} C_VEL
LIN {X 0,Y 340.731,Z 277.852,A -85,B 0,C 180,E1 -14019.478,E2 -14019.478} C_VEL
LIN {X 0,Y 340.938,Z 277.949,A -85,B 0,C 180,E1 -14022.574,E2 -14022.574} C_VEL
LIN {X 0,Y 340.898,Z 282.041,A -85,B 0,C 180,E1 -14023.631,E2 -14023.631} C_VEL
LIN {X 0,Y 343.508,Z 302.81,A -85,B 0,C 180,E1 -14024.306,E2 -14024.306} C_VEL
LIN {X 0,Y 342.283,Z 360.958,A -85,B 0,C 180,E1 -14026.006,E2 -14026.006} C_VEL
LIN {X 0,Y 342.032,Z 371.27,A -85,B 0,C 180,E1 -14026.488,E2 -14026.488} C_VEL
LIN {X 0,Y 341.648,Z 382.685,A -85,B 0,C 180,E1 -14027.229,E2 -14027.229} C_VEL
LIN {X 0,Y 341.286,Z 392.768,A -85,B 0,C 180,E1 -14028.121,E2 -14028.121} C_VEL
LIN {X 0,Y 340.879,Z 402.042,A -85,B 0,C 180,E1 -14029.16,E2 -14029.16} C_VEL
LIN {X 0,Y 340.405,Z 409.614,A -85,B 0,C 180,E1 -14030.197,E2 -14030.197} C_VEL
LIN {X 0,Y 339.966,Z 418.423,A -85,B 0,C 180,E1 -14031.684,E2 -14031.684} C_VEL
LIN {X 0,Y 339.742,Z 424.067,A -85,B 0,C 180,E1 -14032.874,E2 -14032.874} C_VEL
LIN {X 0,Y 339.496,Z 428.775,A -85,B 0,C 180,E1 -14034.063,E2 -14034.063} C_VEL
LIN {X 0,Y 339.449,Z 432.692,A -85,B 0,C 180,E1 -14035.254,E2 -14035.254} C_VEL
LIN {X 0,Y 339.289,Z 435.879,A -85,B 0,C 180,E1 -14036.441,E2 -14036.441} C_VEL
LIN {X 0,Y 339.161,Z 438.384,A -85,B 0,C 180,E1 -14037.629,E2 -14037.629} C_VEL
LIN {X 0,Y 339.139,Z 440.266,A -85,B 0,C 180,E1 -14038.816,E2 -14038.816} C_VEL
LIN {X 0,Y 339.173,Z 441.592,A -85,B 0,C 180,E1 -14040.004,E2 -14040.004} C_VEL
LIN {X 0,Y 339.249,Z 442.385,A -85,B 0,C 180,E1 -14041.191,E2 -14041.191} C_VEL
LIN {X 0,Y 339.419,Z 442.651,A -85,B 0,C 180,E1 -14042.377,E2 -14042.377} C_VEL
LIN {X 0,Y 339.719,Z 442.377,A -85,B 0,C 180,E1 -14043.562,E2 -14043.562} C_VEL
LIN {X 0,Y 340.05,Z 441.503,A -85,B 0,C 180,E1 -14044.746,E2 -14044.746} C_VEL
LIN {X 0,Y 340.287,Z 440.072,A -85,B 0,C 180,E1 -14045.931,E2 -14045.931} C_VEL
LIN {X 0,Y 340.411,Z 438.118,A -85,B 0,C 180,E1 -14047.119,E2 -14047.119} C_VEL
LIN {X 0,Y 341.375,Z 434.213,A -85,B 0,C 180,E1 -14048.811,E2 -14048.811} C_VEL
LIN {X 0,Y 342.176,Z 429.454,A -85,B 0,C 180,E1 -14050.357,E2 -14050.357} C_VEL
LIN {X 0,Y 343.164,Z 423.581,A -85,B 0,C 180,E1 -14051.821,E2 -14051.821} C_VEL
LIN {X 0,Y 344.174,Z 417.857,A -85,B 0,C 180,E1 -14052.984,E2 -14052.984} C_VEL
LIN {X 0,Y 345.19,Z 410.97,A -85,B 0,C 180,E1 -14054.145,E2 -14054.145} C_VEL
LIN {X 0,Y 346.358,Z 402.563,A -85,B 0,C 180,E1 -14055.298,E2 -14055.298} C_VEL
LIN {X 0,Y 347.592,Z 391.94,A -85,B 0,C 180,E1 -14056.447,E2 -14056.447} C_VEL
LIN {X 0,Y 348.548,Z 381.484,A -85,B 0,C 180,E1 -14057.306,E2 -14057.306} C_VEL
LIN {X 0,Y 349.504,Z 369.321,A -85,B 0,C 180,E1 -14058.05,E2 -14058.05} C_VEL
LIN {X 0,Y 350.234,Z 356.917,A -85,B 0,C 180,E1 -14058.541,E2 -14058.541} C_VEL
LIN {X 0,Y 352.814,Z 309.207,A -85,B 0,C 180,E1 -14060.101,E2 -14060.101} C_VEL
LIN {X 0,Y 350.967,Z 301.947,A -85,B 0,C 180,E1 -14060.608,E2 -14060.608} C_VEL
LIN {X 0,Y 346.451,Z 292.325,A -85,B 0,C 180,E1 -14061.579,E2 -14061.579} C_VEL
LIN {X 0,Y 342.99,Z 285.793,A -85,B 0,C 180,E1 -14062.353,E2 -14062.353} C_VEL
LIN {X 0,Y 340.719,Z 277.858,A -85,B 0,C 180,E1 -14065.188,E2 -14065.188} C_VEL
LIN {X 0,Y 340.693,Z 277.858,A -85,B 0,C 180,E1 -14068.327,E2 -14068.327} C_VEL
LIN {X 0,Y 340.703,Z 277.86,A -85,B 0,C 180,E1 -14071.047,E2 -14071.047} C_VEL
LIN {X 0,Y 340.725,Z 277.855,A -85,B 0,C 180,E1 -14075.281,E2 -14075.281} C_VEL
LIN {X 0,Y 340.703,Z 277.86,A -85,B 0,C 180,E1 -14078.384,E2 -14078.384} C_VEL
LIN {X 0,Y 340.704,Z 277.857,A -85,B 0,C 180,E1 -14082.046,E2 -14082.046} C_VEL
LIN {X 0,Y 340.662,Z 277.861,A -85,B 0,C 180,E1 -14086.228,E2 -14086.228} C_VEL
LIN {X 0,Y 340.686,Z 277.859,A -85,B 0,C 180,E1 -14089.757,E2 -14089.757} C_VEL
LIN {X 0,Y 340.712,Z 277.851,A -85,B 0,C 180,E1 -14093.259,E2 -14093.259} C_VEL
LIN {X 0,Y 340.703,Z 277.853,A -85,B 0,C 180,E1 -14096.154,E2 -14096.154} C_VEL
LIN {X 0,Y 340.748,Z 277.85,A -85,B 0,C 180,E1 -14100.33,E2 -14100.33} C_VEL
LIN {X 0,Y 340.868,Z 277.952,A -85,B 0,C 180,E1 -14103.232,E2 -14103.232} C_VEL
LIN {X 0,Y 342.612,Z 288.19,A -85,B 0,C 180,E1 -14106.1,E2 -14106.1} C_VEL
LIN {X 0,Y 342.66,Z 289.928,A -85,B 0,C 180,E1 -14106.545,E2 -14106.545} C_VEL
LIN {X 0,Y 344.019,Z 301.172,A -85,B 0,C 180,E1 -14107.845,E2 -14107.845} C_VEL
LIN {X 0,Y 346.624,Z 313.571,A -85,B 0,C 180,E1 -14108.717,E2 -14108.717} C_VEL
LIN {X 0,Y 349.727,Z 333.791,A -85,B 0,C 180,E1 -14109.909,E2 -14109.909} C_VEL
LIN {X 0,Y 350.755,Z 347.228,A -85,B 0,C 180,E1 -14110.563,E2 -14110.563} C_VEL
LIN {X 0,Y 348.531,Z 392.448,A -85,B 0,C 180,E1 -14112.084,E2 -14112.084} C_VEL
LIN {X 0,Y 347.387,Z 404.69,A -85,B 0,C 180,E1 -14112.714,E2 -14112.714} C_VEL
LIN {X 0,Y 346.391,Z 413.604,A -85,B 0,C 180,E1 -14113.346,E2 -14113.346} C_VEL
LIN {X 0,Y 345.166,Z 423.09,A -85,B 0,C 180,E1 -14114.197,E2 -14114.197} C_VEL
LIN {X 0,Y 343.824,Z 433.181,A -85,B 0,C 180,E1 -14115.347,E2 -14115.347} C_VEL
LIN {X 0,Y 342.605,Z 441.991,A -85,B 0,C 180,E1 -14116.657,E2 -14116.657} C_VEL
LIN {X 0,Y 341.667,Z 448.444,A -85,B 0,C 180,E1 -14117.828,E2 -14117.828} C_VEL
LIN {X 0,Y 340.877,Z 453.834,A -85,B 0,C 180,E1 -14119.005,E2 -14119.005} C_VEL
LIN {X 0,Y 340.184,Z 459.372,A -85,B 0,C 180,E1 -14120.487,E2 -14120.487} C_VEL
LIN {X 0,Y 339.569,Z 464.538,A -85,B 0,C 180,E1 -14122.268,E2 -14122.268} C_VEL
LIN {X 0,Y 339.199,Z 468.11,A -85,B 0,C 180,E1 -14124.053,E2 -14124.053} C_VEL
LIN {X 0,Y 339.151,Z 469.834,A -85,B 0,C 180,E1 -14125.245,E2 -14125.245} C_VEL
LIN {X 0,Y 339.206,Z 472.844,A -85,B 0,C 180,E1 -14128.813,E2 -14128.813} C_VEL
LIN {X 0,Y 339.228,Z 473.476,A -85,B 0,C 180,E1 -14130,E2 -14130} C_VEL
LIN {X 0,Y 339.144,Z 473.638,A -85,B 0,C 180,E1 -14131.187,E2 -14131.187} C_VEL
LIN {X 0,Y 339.076,Z 473.279,A -85,B 0,C 180,E1 -14132.376,E2 -14132.376} C_VEL
LIN {X 0,Y 339.117,Z 472.344,A -85,B 0,C 180,E1 -14133.564,E2 -14133.564} C_VEL
LIN {X 0,Y 339.146,Z 470.929,A -85,B 0,C 180,E1 -14134.755,E2 -14134.755} C_VEL
LIN {X 0,Y 339.289,Z 467.848,A -85,B 0,C 180,E1 -14136.541,E2 -14136.541} C_VEL
LIN {X 0,Y 339.717,Z 463.494,A -85,B 0,C 180,E1 -14138.326,E2 -14138.326} C_VEL
LIN {X 0,Y 340.4,Z 457.494,A -85,B 0,C 180,E1 -14140.107,E2 -14140.107} C_VEL
LIN {X 0,Y 341,Z 452.551,A -85,B 0,C 180,E1 -14141.291,E2 -14141.291} C_VEL
LIN {X 0,Y 341.78,Z 446.611,A -85,B 0,C 180,E1 -14142.469,E2 -14142.469} C_VEL
LIN {X 0,Y 342.701,Z 439.401,A -85,B 0,C 180,E1 -14143.641,E2 -14143.641} C_VEL
LIN {X 0,Y 343.682,Z 431.719,A -85,B 0,C 180,E1 -14144.658,E2 -14144.658} C_VEL
LIN {X 0,Y 344.545,Z 423.671,A -85,B 0,C 180,E1 -14145.529,E2 -14145.529} C_VEL
LIN {X 0,Y 345.357,Z 415.346,A -85,B 0,C 180,E1 -14146.249,E2 -14146.249} C_VEL
LIN {X 0,Y 346.066,Z 406.872,A -85,B 0,C 180,E1 -14146.821,E2 -14146.821} C_VEL
LIN {X 0,Y 346.816,Z 396.798,A -85,B 0,C 180,E1 -14147.315,E2 -14147.315} C_VEL
LIN {X 0,Y 347.362,Z 383.838,A -85,B 0,C 180,E1 -14147.7,E2 -14147.7} C_VEL
LIN {X 0,Y 347.849,Z 345.649,A -85,B 0,C 180,E1 -14148.516,E2 -14148.516} C_VEL
LIN {X 0,Y 344.972,Z 326.191,A -85,B 0,C 180,E1 -14149.151,E2 -14149.151} C_VEL
LIN {X 0,Y 342.286,Z 312.063,A -85,B 0,C 180,E1 -14149.687,E2 -14149.687} C_VEL
LIN {X 0,Y 343.857,Z 296.639,A -85,B 0,C 180,E1 -14153.807,E2 -14153.807} C_VEL
LIN {X 0,Y 343.817,Z 293.179,A -85,B 0,C 180,E1 -14154.774,E2 -14154.774} C_VEL
LIN {X 0,Y 342.27,Z 284.585,A -85,B 0,C 180,E1 -14157.346,E2 -14157.346} C_VEL
LIN {X 0,Y 340.743,Z 277.85,A -85,B 0,C 180,E1 -14159.5,E2 -14159.5} C_VEL
LIN {X 0,Y 340.695,Z 277.852,A -85,B 0,C 180,E1 -14162.435,E2 -14162.435} C_VEL
LIN {X 0,Y 340.724,Z 277.848,A -85,B 0,C 180,E1 -14165.278,E2 -14165.278} C_VEL
LIN {X 0,Y 340.702,Z 277.857,A -85,B 0,C 180,E1 -14168.381,E2 -14168.381} C_VEL
LIN {X 0,Y 340.706,Z 277.857,A -85,B 0,C 180,E1 -14172.043,E2 -14172.043} C_VEL
LIN {X 0,Y 340.66,Z 277.862,A -85,B 0,C 180,E1 -14176.225,E2 -14176.225} C_VEL
LIN {X 0,Y 340.68,Z 277.859,A -85,B 0,C 180,E1 -14178.686,E2 -14178.686} C_VEL
LIN {X 0,Y 340.727,Z 277.853,A -85,B 0,C 180,E1 -14181.769,E2 -14181.769} C_VEL
LIN {X 0,Y 340.731,Z 277.85,A -85,B 0,C 180,E1 -14185.593,E2 -14185.593} C_VEL
LIN {X 0,Y 340.701,Z 277.85,A -85,B 0,C 180,E1 -14188.952,E2 -14188.952} C_VEL
LIN {X 0,Y 340.732,Z 277.849,A -85,B 0,C 180,E1 -14193.011,E2 -14193.011} C_VEL
LIN {X 0,Y 340.762,Z 277.851,A -85,B 0,C 180,E1 -14195.636,E2 -14195.636} C_VEL
LIN {X 0,Y 340.736,Z 277.845,A -85,B 0,C 180,E1 -14199.47,E2 -14199.47} C_VEL
LIN {X 0,Y 340.798,Z 277.843,A -85,B 0,C 180,E1 -14201.978,E2 -14201.978} C_VEL
LIN {X 0,Y 340.874,Z 277.833,A -85,B 0,C 180,E1 -14205.702,E2 -14205.702} C_VEL
LIN {X 0,Y 340.874,Z 277.822,A -85,B 0,C 180,E1 -14209.303,E2 -14209.303} C_VEL
LIN {X 0,Y 341.061,Z 277.805,A -85,B 0,C 180,E1 -14212.894,E2 -14212.894} C_VEL
LIN {X 0,Y 341.157,Z 277.797,A -85,B 0,C 180,E1 -14217.635,E2 -14217.635} C_VEL
LIN {X 0,Y 341.254,Z 277.777,A -85,B 0,C 180,E1 -14219.996,E2 -14219.996} C_VEL
LIN {X 0,Y 341.164,Z 277.799,A -85,B 0,C 180,E1 -14222.357,E2 -14222.357} C_VEL
LIN {X 0,Y 341.012,Z 277.815,A -85,B 0,C 180,E1 -14227.099,E2 -14227.099} C_VEL
LIN {X 0,Y 340.843,Z 277.832,A -85,B 0,C 180,E1 -14230.69,E2 -14230.69} C_VEL
LIN {X 0,Y 340.857,Z 277.836,A -85,B 0,C 180,E1 -14234.321,E2 -14234.321} C_VEL
LIN {X 0,Y 340.829,Z 277.843,A -85,B 0,C 180,E1 -14238.462,E2 -14238.462} C_VEL
LIN {X 0,Y 340.743,Z 277.85,A -85,B 0,C 180,E1 -14241.853,E2 -14241.853} C_VEL
LIN {X 0,Y 340.76,Z 277.847,A -85,B 0,C 180,E1 -14245.66,E2 -14245.66} C_VEL
LIN {X 0,Y 340.714,Z 277.854,A -85,B 0,C 180,E1 -14248.317,E2 -14248.317} C_VEL
LIN {X 0,Y 340.682,Z 277.857,A -85,B 0,C 180,E1 -14251.041,E2 -14251.041} C_VEL
LIN {X 0,Y 340.7,Z 277.846,A -85,B 0,C 180,E1 -14255.275,E2 -14255.275} C_VEL
LIN {X 0,Y 340.692,Z 277.862,A -85,B 0,C 180,E1 -14258.382,E2 -14258.382} C_VEL
LIN {X 0,Y 340.704,Z 277.855,A -85,B 0,C 180,E1 -14261.3,E2 -14261.3} C_VEL
LIN {X 0,Y 340.759,Z 277.847,A -85,B 0,C 180,E1 -14264.519,E2 -14264.519} C_VEL
LIN {X 0,Y 340.727,Z 277.855,A -85,B 0,C 180,E1 -14267.941,E2 -14267.941} C_VEL
LIN {X 0,Y 340.724,Z 277.902,A -85,B 0,C 180,E1 -14271.433,E2 -14271.433} C_VEL
LIN {X 0,Y 341.948,Z 283.661,A -85,B 0,C 180,E1 -14273.338,E2 -14273.338} C_VEL
LIN {X 0,Y 346.397,Z 295.545,A -85,B 0,C 180,E1 -14273.938,E2 -14273.938} C_VEL
LIN {X 0,Y 348.714,Z 306.03,A -85,B 0,C 180,E1 -14274.339,E2 -14274.339} C_VEL
LIN {X 0,Y 347.588,Z 360.681,A -85,B 0,C 180,E1 -14275.519,E2 -14275.519} C_VEL
LIN {X 0,Y 347.2,Z 371.234,A -85,B 0,C 180,E1 -14275.93,E2 -14275.93} C_VEL
LIN {X 0,Y 346.491,Z 383.596,A -85,B 0,C 180,E1 -14276.692,E2 -14276.692} C_VEL
LIN {X 0,Y 345.749,Z 392.135,A -85,B 0,C 180,E1 -14277.408,E2 -14277.408} C_VEL
LIN {X 0,Y 344.96,Z 400.618,A -85,B 0,C 180,E1 -14278.312,E2 -14278.312} C_VEL
LIN {X 0,Y 344.095,Z 408.136,A -85,B 0,C 180,E1 -14279.295,E2 -14279.295} C_VEL
LIN {X 0,Y 343.318,Z 414.129,A -85,B 0,C 180,E1 -14280.237,E2 -14280.237} C_VEL
LIN {X 0,Y 342.606,Z 419.252,A -85,B 0,C 180,E1 -14281.18,E2 -14281.18} C_VEL
LIN {X 0,Y 341.813,Z 425.403,A -85,B 0,C 180,E1 -14282.564,E2 -14282.564} C_VEL
LIN {X 0,Y 341.037,Z 430.638,A -85,B 0,C 180,E1 -14284.029,E2 -14284.029} C_VEL
LIN {X 0,Y 340.378,Z 435.05,A -85,B 0,C 180,E1 -14285.61,E2 -14285.61} C_VEL
LIN {X 0,Y 339.792,Z 438.926,A -85,B 0,C 180,E1 -14287.503,E2 -14287.503} C_VEL
LIN {X 0,Y 339.377,Z 441.276,A -85,B 0,C 180,E1 -14289.388,E2 -14289.388} C_VEL
LIN {X 0,Y 339.168,Z 442.203,A -85,B 0,C 180,E1 -14290.638,E2 -14290.638} C_VEL
LIN {X 0,Y 339.035,Z 442.458,A -85,B 0,C 180,E1 -14292.45,E2 -14292.45} C_VEL
LIN {X 0,Y 339.033,Z 441.497,A -85,B 0,C 180,E1 -14294.367,E2 -14294.367} C_VEL
LIN {X 0,Y 339.144,Z 440.211,A -85,B 0,C 180,E1 -14295.601,E2 -14295.601} C_VEL
LIN {X 0,Y 339.294,Z 438.39,A -85,B 0,C 180,E1 -14296.83,E2 -14296.83} C_VEL
LIN {X 0,Y 339.472,Z 435.979,A -85,B 0,C 180,E1 -14298.052,E2 -14298.052} C_VEL
LIN {X 0,Y 339.817,Z 431.045,A -85,B 0,C 180,E1 -14299.875,E2 -14299.875} C_VEL
LIN {X 0,Y 340.142,Z 426.913,A -85,B 0,C 180,E1 -14301.085,E2 -14301.085} C_VEL
LIN {X 0,Y 340.525,Z 421.337,A -85,B 0,C 180,E1 -14302.415,E2 -14302.415} C_VEL
LIN {X 0,Y 340.963,Z 415.91,A -85,B 0,C 180,E1 -14303.491,E2 -14303.491} C_VEL
LIN {X 0,Y 341.55,Z 408.56,A -85,B 0,C 180,E1 -14304.687,E2 -14304.687} C_VEL
LIN {X 0,Y 342.032,Z 401.958,A -85,B 0,C 180,E1 -14305.581,E2 -14305.581} C_VEL
LIN {X 0,Y 342.602,Z 393.94,A -85,B 0,C 180,E1 -14306.472,E2 -14306.472} C_VEL
LIN {X 0,Y 343.075,Z 385.679,A -85,B 0,C 180,E1 -14307.212,E2 -14307.212} C_VEL
LIN {X 0,Y 343.437,Z 377.333,A -85,B 0,C 180,E1 -14307.801,E2 -14307.801} C_VEL
LIN {X 0,Y 343.78,Z 368.288,A -85,B 0,C 180,E1 -14308.28,E2 -14308.28} C_VEL
LIN {X 0,Y 343.981,Z 359.205,A -85,B 0,C 180,E1 -14308.61,E2 -14308.61} C_VEL
LIN {X 0,Y 344.81,Z 303.835,A -85,B 0,C 180,E1 -14309.789,E2 -14309.789} C_VEL
LIN {X 0,Y 341.481,Z 283.172,A -85,B 0,C 180,E1 -14310.369,E2 -14310.369} C_VEL
LIN {X 0,Y 341.137,Z 277.852,A -85,B 0,C 180,E1 -14311.993,E2 -14311.993} C_VEL
LIN {X 0,Y 341.025,Z 277.82,A -85,B 0,C 180,E1 -14317.103,E2 -14317.103} C_VEL
LIN {X 0,Y 340.836,Z 277.839,A -85,B 0,C 180,E1 -14320.695,E2 -14320.695} C_VEL
LIN {X 0,Y 340.83,Z 277.839,A -85,B 0,C 180,E1 -14324.326,E2 -14324.326} C_VEL
LIN {X 0,Y 340.805,Z 277.842,A -85,B 0,C 180,E1 -14328.468,E2 -14328.468} C_VEL
LIN {X 0,Y 340.723,Z 277.854,A -85,B 0,C 180,E1 -14331.859,E2 -14331.859} C_VEL
LIN {X 0,Y 340.69,Z 277.86,A -85,B 0,C 180,E1 -14335.671,E2 -14335.671} C_VEL
LIN {X 0,Y 340.676,Z 277.862,A -85,B 0,C 180,E1 -14339.677,E2 -14339.677} C_VEL
LIN {X 0,Y 340.66,Z 277.862,A -85,B 0,C 180,E1 -14343.776,E2 -14343.776} C_VEL
LIN {X 0,Y 340.046,Z 277.945,A -85,B 0,C 180,E1 -14344.763,E2 -14344.763} C_VEL
LIN {X 0,Y 337.199,Z 278.297,A -85,B 0,C 180,E1 -14346.368,E2 -14346.368} C_VEL
LIN {X 0,Y 334.743,Z 278.603,A -85,B 0,C 180,E1 -14347.668,E2 -14347.668} C_VEL
LIN {X 0,Y 333.674,Z 278.731,A -85,B 0,C 180,E1 -14348.675,E2 -14348.675} C_VEL
LIN {X 0,Y 333.581,Z 278.742,A -85,B 0,C 180,E1 -14349.016,E2 -14349.016} C_VEL
LIN {X 0,Y 333.606,Z 278.739,A -85,B 0,C 180,E1 -14352.503,E2 -14352.503} C_VEL
LIN {X 0,Y 333.575,Z 278.746,A -85,B 0,C 180,E1 -14355.959,E2 -14355.959} C_VEL
LIN {X 0,Y 333.628,Z 278.738,A -85,B 0,C 180,E1 -14359.32,E2 -14359.32} C_VEL
LIN {X 0,Y 333.648,Z 278.734,A -85,B 0,C 180,E1 -14363.172,E2 -14363.172} C_VEL
LIN {X 0,Y 333.658,Z 278.733,A -85,B 0,C 180,E1 -14365.346,E2 -14365.346} C_VEL
LIN {X 0,Y 333.615,Z 278.74,A -85,B 0,C 180,E1 -14368.226,E2 -14368.226} C_VEL
LIN {X 0,Y 333.641,Z 278.734,A -85,B 0,C 180,E1 -14371.027,E2 -14371.027} C_VEL
LIN {X 0,Y 333.687,Z 278.729,A -85,B 0,C 180,E1 -14375.093,E2 -14375.093} C_VEL
LIN {X 0,Y 333.668,Z 278.731,A -85,B 0,C 180,E1 -14379.023,E2 -14379.023} C_VEL
LIN {X 0,Y 333.894,Z 278.74,A -85,B 0,C 180,E1 -14382.551,E2 -14382.551} C_VEL
LIN {X 0,Y 333.854,Z 282.097,A -85,B 0,C 180,E1 -14383.46,E2 -14383.46} C_VEL
LIN {X 0,Y 336.361,Z 301.905,A -85,B 0,C 180,E1 -14384.124,E2 -14384.124} C_VEL
LIN {X 0,Y 335.209,Z 361.397,A -85,B 0,C 180,E1 -14385.936,E2 -14385.936} C_VEL
LIN {X 0,Y 334.951,Z 371.646,A -85,B 0,C 180,E1 -14386.428,E2 -14386.428} C_VEL
LIN {X 0,Y 334.557,Z 383.029,A -85,B 0,C 180,E1 -14387.185,E2 -14387.185} C_VEL
LIN {X 0,Y 334.184,Z 393.825,A -85,B 0,C 180,E1 -14388.172,E2 -14388.172} C_VEL
LIN {X 0,Y 333.701,Z 402.976,A -85,B 0,C 180,E1 -14389.232,E2 -14389.232} C_VEL
LIN {X 0,Y 333.179,Z 412.441,A -85,B 0,C 180,E1 -14390.596,E2 -14390.596} C_VEL
LIN {X 0,Y 332.857,Z 419.147,A -85,B 0,C 180,E1 -14391.81,E2 -14391.81} C_VEL
LIN {X 0,Y 332.587,Z 425.008,A -85,B 0,C 180,E1 -14393.094,E2 -14393.094} C_VEL
LIN {X 0,Y 332.373,Z 430.402,A -85,B 0,C 180,E1 -14394.544,E2 -14394.544} C_VEL
LIN {X 0,Y 332.311,Z 434.078,A -85,B 0,C 180,E1 -14395.759,E2 -14395.759} C_VEL
LIN {X 0,Y 332.074,Z 438.304,A -85,B 0,C 180,E1 -14397.578,E2 -14397.578} C_VEL
LIN {X 0,Y 332.041,Z 440.305,A -85,B 0,C 180,E1 -14398.791,E2 -14398.791} C_VEL
LIN {X 0,Y 332.075,Z 441.753,A -85,B 0,C 180,E1 -14400.004,E2 -14400.004} C_VEL
LIN {X 0,Y 332.157,Z 442.671,A -85,B 0,C 180,E1 -14401.216,E2 -14401.216} C_VEL
LIN {X 0,Y 332.337,Z 443.06,A -85,B 0,C 180,E1 -14402.428,E2 -14402.428} C_VEL
LIN {X 0,Y 332.648,Z 442.843,A -85,B 0,C 180,E1 -14403.638,E2 -14403.638} C_VEL
LIN {X 0,Y 333.005,Z 442.048,A -85,B 0,C 180,E1 -14404.846,E2 -14404.846} C_VEL
LIN {X 0,Y 333.255,Z 440.742,A -85,B 0,C 180,E1 -14406.056,E2 -14406.056} C_VEL
LIN {X 0,Y 333.418,Z 438.908,A -85,B 0,C 180,E1 -14407.269,E2 -14407.269} C_VEL
LIN {X 0,Y 334.218,Z 436.436,A -85,B 0,C 180,E1 -14408.468,E2 -14408.468} C_VEL
LIN {X 0,Y 334.702,Z 433.402,A -85,B 0,C 180,E1 -14409.674,E2 -14409.674} C_VEL
LIN {X 0,Y 335.733,Z 428.491,A -85,B 0,C 180,E1 -14411.168,E2 -14411.168} C_VEL
LIN {X 0,Y 336.862,Z 422.33,A -85,B 0,C 180,E1 -14412.657,E2 -14412.657} C_VEL
LIN {X 0,Y 338.199,Z 414.658,A -85,B 0,C 180,E1 -14414.136,E2 -14414.136} C_VEL
LIN {X 0,Y 339.531,Z 405.833,A -85,B 0,C 180,E1 -14415.46,E2 -14415.46} C_VEL
LIN {X 0,Y 340.698,Z 397.428,A -85,B 0,C 180,E1 -14416.481,E2 -14416.481} C_VEL
LIN {X 0,Y 341.746,Z 388.588,A -85,B 0,C 180,E1 -14417.352,E2 -14417.352} C_VEL
LIN {X 0,Y 342.844,Z 377.154,A -85,B 0,C 180,E1 -14418.22,E2 -14418.22} C_VEL
LIN {X 0,Y 343.601,Z 367.259,A -85,B 0,C 180,E1 -14418.758,E2 -14418.758} C_VEL
LIN {X 0,Y 344.355,Z 354.864,A -85,B 0,C 180,E1 -14419.225,E2 -14419.225} C_VEL
LIN {X 0,Y 346.929,Z 310.774,A -85,B 0,C 180,E1 -14420.727,E2 -14420.727} C_VEL
LIN {X 0,Y 345.493,Z 305.062,A -85,B 0,C 180,E1 -14421.151,E2 -14421.151} C_VEL
LIN {X 0,Y 340.665,Z 294.893,A -85,B 0,C 180,E1 -14422.243,E2 -14422.243} C_VEL
LIN {X 0,Y 335.947,Z 286.295,A -85,B 0,C 180,E1 -14423.356,E2 -14423.356} C_VEL
LIN {X 0,Y 333.646,Z 278.737,A -85,B 0,C 180,E1 -14426.257,E2 -14426.257} C_VEL
LIN {X 0,Y 333.663,Z 278.737,A -85,B 0,C 180,E1 -14428.98,E2 -14428.98} C_VEL
LIN {X 0,Y 333.653,Z 278.738,A -85,B 0,C 180,E1 -14432.589,E2 -14432.589} C_VEL
LIN {X 0,Y 333.683,Z 278.734,A -85,B 0,C 180,E1 -14436.141,E2 -14436.141} C_VEL
LIN {X 0,Y 333.612,Z 278.741,A -85,B 0,C 180,E1 -14439.201,E2 -14439.201} C_VEL
LIN {X 0,Y 333.639,Z 278.738,A -85,B 0,C 180,E1 -14442.501,E2 -14442.501} C_VEL
LIN {X 0,Y 333.606,Z 278.74,A -85,B 0,C 180,E1 -14445.956,E2 -14445.956} C_VEL
LIN {X 0,Y 333.654,Z 278.736,A -85,B 0,C 180,E1 -14449.318,E2 -14449.318} C_VEL
LIN {X 0,Y 333.673,Z 278.728,A -85,B 0,C 180,E1 -14453.17,E2 -14453.17} C_VEL
LIN {X 0,Y 333.684,Z 278.731,A -85,B 0,C 180,E1 -14455.342,E2 -14455.342} C_VEL
LIN {X 0,Y 333.7,Z 278.732,A -85,B 0,C 180,E1 -14459.638,E2 -14459.638} C_VEL
LIN {X 0,Y 333.846,Z 278.894,A -85,B 0,C 180,E1 -14463.088,E2 -14463.088} C_VEL
LIN {X 0,Y 334.798,Z 284.156,A -85,B 0,C 180,E1 -14464.591,E2 -14464.591} C_VEL
LIN {X 0,Y 336.956,Z 292.8,A -85,B 0,C 180,E1 -14466.002,E2 -14466.002} C_VEL
LIN {X 0,Y 337.85,Z 300.841,A -85,B 0,C 180,E1 -14466.976,E2 -14466.976} C_VEL
LIN {X 0,Y 340.626,Z 313.702,A -85,B 0,C 180,E1 -14467.951,E2 -14467.951} C_VEL
LIN {X 0,Y 343.501,Z 332.617,A -85,B 0,C 180,E1 -14469.155,E2 -14469.155} C_VEL
LIN {X 0,Y 344.619,Z 345.012,A -85,B 0,C 180,E1 -14469.798,E2 -14469.798} C_VEL
LIN {X 0,Y 344.737,Z 351.622,A -85,B 0,C 180,E1 -14470.085,E2 -14470.085} C_VEL
LIN {X 0,Y 342.311,Z 392.923,A -85,B 0,C 180,E1 -14471.521,E2 -14471.521} C_VEL
LIN {X 0,Y 341.123,Z 404.685,A -85,B 0,C 180,E1 -14472.154,E2 -14472.154} C_VEL
LIN {X 0,Y 339.947,Z 414.399,A -85,B 0,C 180,E1 -14472.866,E2 -14472.866} C_VEL
LIN {X 0,Y 338.484,Z 425.059,A -85,B 0,C 180,E1 -14473.876,E2 -14473.876} C_VEL
LIN {X 0,Y 337.06,Z 434.417,A -85,B 0,C 180,E1 -14475.047,E2 -14475.047} C_VEL
LIN {X 0,Y 336.043,Z 441.181,A -85,B 0,C 180,E1 -14476.083,E2 -14476.083} C_VEL
LIN {X 0,Y 335.094,Z 447.697,A -85,B 0,C 180,E1 -14477.278,E2 -14477.278} C_VEL
LIN {X 0,Y 334.142,Z 453.159,A -85,B 0,C 180,E1 -14478.474,E2 -14478.474} C_VEL
LIN {X 0,Y 333.373,Z 458.738,A -85,B 0,C 180,E1 -14479.984,E2 -14479.984} C_VEL
LIN {X 0,Y 332.719,Z 463.155,A -85,B 0,C 180,E1 -14481.497,E2 -14481.497} C_VEL
LIN {X 0,Y 332.228,Z 467.124,A -85,B 0,C 180,E1 -14483.318,E2 -14483.318} C_VEL
LIN {X 0,Y 332.055,Z 469.661,A -85,B 0,C 180,E1 -14485.143,E2 -14485.143} C_VEL
LIN {X 0,Y 332.058,Z 470.73,A -85,B 0,C 180,E1 -14486.359,E2 -14486.359} C_VEL
LIN {X 0,Y 332.031,Z 471.312,A -85,B 0,C 180,E1 -14487.574,E2 -14487.574} C_VEL
LIN {X 0,Y 332.11,Z 472.449,A -85,B 0,C 180,E1 -14488.787,E2 -14488.787} C_VEL
LIN {X 0,Y 332.136,Z 473.126,A -85,B 0,C 180,E1 -14490,E2 -14490} C_VEL
LIN {X 0,Y 332.046,Z 473.33,A -85,B 0,C 180,E1 -14491.213,E2 -14491.213} C_VEL
LIN {X 0,Y 331.989,Z 472.978,A -85,B 0,C 180,E1 -14492.426,E2 -14492.426} C_VEL
LIN {X 0,Y 332.042,Z 472.081,A -85,B 0,C 180,E1 -14493.64,E2 -14493.64} C_VEL
LIN {X 0,Y 332.085,Z 469.178,A -85,B 0,C 180,E1 -14495.899,E2 -14495.899} C_VEL
LIN {X 0,Y 332.364,Z 466.444,A -85,B 0,C 180,E1 -14497.289,E2 -14497.289} C_VEL
LIN {X 0,Y 332.866,Z 461.547,A -85,B 0,C 180,E1 -14499.111,E2 -14499.111} C_VEL
LIN {X 0,Y 333.532,Z 456.303,A -85,B 0,C 180,E1 -14500.624,E2 -14500.624} C_VEL
LIN {X 0,Y 334.244,Z 451.184,A -85,B 0,C 180,E1 -14501.83,E2 -14501.83} C_VEL
LIN {X 0,Y 335.072,Z 445.047,A -85,B 0,C 180,E1 -14503.031,E2 -14503.031} C_VEL
LIN {X 0,Y 335.927,Z 438.62,A -85,B 0,C 180,E1 -14504.076,E2 -14504.076} C_VEL
LIN {X 0,Y 336.974,Z 430.856,A -85,B 0,C 180,E1 -14505.112,E2 -14505.112} C_VEL
LIN {X 0,Y 337.748,Z 424.193,A -85,B 0,C 180,E1 -14505.849,E2 -14505.849} C_VEL
LIN {X 0,Y 338.592,Z 416.089,A -85,B 0,C 180,E1 -14506.583,E2 -14506.583} C_VEL
LIN {X 0,Y 339.41,Z 406.739,A -85,B 0,C 180,E1 -14507.239,E2 -14507.239} C_VEL
LIN {X 0,Y 340.215,Z 396.744,A -85,B 0,C 180,E1 -14507.74,E2 -14507.74} C_VEL
LIN {X 0,Y 340.74,Z 384.578,A -85,B 0,C 180,E1 -14508.124,E2 -14508.124} C_VEL
LIN {X 0,Y 341.309,Z 346.627,A -85,B 0,C 180,E1 -14508.947,E2 -14508.947} C_VEL
LIN {X 0,Y 338.521,Z 327.628,A -85,B 0,C 180,E1 -14509.584,E2 -14509.584} C_VEL
LIN {X 0,Y 335.477,Z 311.65,A -85,B 0,C 180,E1 -14510.223,E2 -14510.223} C_VEL
LIN {X 0,Y 336.954,Z 297.81,A -85,B 0,C 180,E1 -14513.999,E2 -14513.999} C_VEL
LIN {X 0,Y 336.851,Z 294.363,A -85,B 0,C 180,E1 -14514.992,E2 -14514.992} C_VEL
LIN {X 0,Y 335.409,Z 286.33,A -85,B 0,C 180,E1 -14517.45,E2 -14517.45} C_VEL
LIN {X 0,Y 333.712,Z 278.725,A -85,B 0,C 180,E1 -14519.892,E2 -14519.892} C_VEL
LIN {X 0,Y 333.646,Z 278.734,A -85,B 0,C 180,E1 -14523.207,E2 -14523.207} C_VEL
LIN {X 0,Y 333.682,Z 278.723,A -85,B 0,C 180,E1 -14526.138,E2 -14526.138} C_VEL
LIN {X 0,Y 333.641,Z 278.736,A -85,B 0,C 180,E1 -14529.193,E2 -14529.193} C_VEL
LIN {X 0,Y 333.64,Z 278.737,A -85,B 0,C 180,E1 -14532.498,E2 -14532.498} C_VEL
LIN {X 0,Y 333.604,Z 278.742,A -85,B 0,C 180,E1 -14535.953,E2 -14535.953} C_VEL
LIN {X 0,Y 333.611,Z 278.743,A -85,B 0,C 180,E1 -14539.322,E2 -14539.322} C_VEL
LIN {X 0,Y 333.671,Z 278.734,A -85,B 0,C 180,E1 -14543.166,E2 -14543.166} C_VEL
LIN {X 0,Y 333.682,Z 278.726,A -85,B 0,C 180,E1 -14545.339,E2 -14545.339} C_VEL
LIN {X 0,Y 333.636,Z 278.732,A -85,B 0,C 180,E1 -14548.219,E2 -14548.219} C_VEL
LIN {X 0,Y 333.661,Z 278.733,A -85,B 0,C 180,E1 -14551.02,E2 -14551.02} C_VEL
LIN {X 0,Y 333.715,Z 278.724,A -85,B 0,C 180,E1 -14555.087,E2 -14555.087} C_VEL
LIN {X 0,Y 333.676,Z 278.722,A -85,B 0,C 180,E1 -14559.016,E2 -14559.016} C_VEL
LIN {X 0,Y 333.746,Z 278.725,A -85,B 0,C 180,E1 -14561.583,E2 -14561.583} C_VEL
LIN {X 0,Y 333.813,Z 278.711,A -85,B 0,C 180,E1 -14565.574,E2 -14565.574} C_VEL
LIN {X 0,Y 333.837,Z 278.698,A -85,B 0,C 180,E1 -14569.075,E2 -14569.075} C_VEL
LIN {X 0,Y 334.008,Z 278.684,A -85,B 0,C 180,E1 -14572.744,E2 -14572.744} C_VEL
LIN {X 0,Y 333.799,Z 278.704,A -85,B 0,C 180,E1 -14575.165,E2 -14575.165} C_VEL
LIN {X 0,Y 334.094,Z 278.676,A -85,B 0,C 180,E1 -14577.585,E2 -14577.585} C_VEL
LIN {X 0,Y 334.206,Z 278.655,A -85,B 0,C 180,E1 -14579.996,E2 -14579.996} C_VEL
LIN {X 0,Y 334.101,Z 278.678,A -85,B 0,C 180,E1 -14582.407,E2 -14582.407} C_VEL
LIN {X 0,Y 333.965,Z 278.687,A -85,B 0,C 180,E1 -14586.516,E2 -14586.516} C_VEL
LIN {X 0,Y 333.816,Z 278.712,A -85,B 0,C 180,E1 -14589.692,E2 -14589.692} C_VEL
LIN {X 0,Y 333.791,Z 278.717,A -85,B 0,C 180,E1 -14593.387,E2 -14593.387} C_VEL
LIN {X 0,Y 333.739,Z 278.722,A -85,B 0,C 180,E1 -14597.142,E2 -14597.142} C_VEL
LIN {X 0,Y 333.728,Z 278.723,A -85,B 0,C 180,E1 -14599.686,E2 -14599.686} C_VEL
LIN {X 0,Y 333.682,Z 278.733,A -85,B 0,C 180,E1 -14602.274,E2 -14602.274} C_VEL
LIN {X 0,Y 333.722,Z 278.727,A -85,B 0,C 180,E1 -14606.242,E2 -14606.242} C_VEL
LIN {X 0,Y 333.676,Z 278.732,A -85,B 0,C 180,E1 -14608.97,E2 -14608.97} C_VEL
LIN {X 0,Y 333.627,Z 278.739,A -85,B 0,C 180,E1 -14612.583,E2 -14612.583} C_VEL
LIN {X 0,Y 333.658,Z 278.721,A -85,B 0,C 180,E1 -14616.135,E2 -14616.135} C_VEL
LIN {X 0,Y 333.662,Z 278.732,A -85,B 0,C 180,E1 -14619.183,E2 -14619.183} C_VEL
LIN {X 0,Y 333.682,Z 278.737,A -85,B 0,C 180,E1 -14622.509,E2 -14622.509} C_VEL
LIN {X 0,Y 333.706,Z 278.731,A -85,B 0,C 180,E1 -14625.973,E2 -14625.973} C_VEL
LIN {X 0,Y 333.677,Z 278.731,A -85,B 0,C 180,E1 -14629.301,E2 -14629.301} C_VEL
LIN {X 0,Y 333.703,Z 278.899,A -85,B 0,C 180,E1 -14631.055,E2 -14631.055} C_VEL
LIN {X 0,Y 334.85,Z 284.251,A -85,B 0,C 180,E1 -14632.802,E2 -14632.802} C_VEL
LIN {X 0,Y 340.012,Z 297.329,A -85,B 0,C 180,E1 -14633.508,E2 -14633.508} C_VEL
LIN {X 0,Y 342.144,Z 306.769,A -85,B 0,C 180,E1 -14633.883,E2 -14633.883} C_VEL
LIN {X 0,Y 341.052,Z 360.023,A -85,B 0,C 180,E1 -14635.05,E2 -14635.05} C_VEL
LIN {X 0,Y 340.713,Z 369.539,A -85,B 0,C 180,E1 -14635.407,E2 -14635.407} C_VEL
LIN {X 0,Y 340.19,Z 379.436,A -85,B 0,C 180,E1 -14635.958,E2 -14635.958} C_VEL
LIN {X 0,Y 339.414,Z 389.518,A -85,B 0,C 180,E1 -14636.721,E2 -14636.721} C_VEL
LIN {X 0,Y 338.47,Z 398.961,A -85,B 0,C 180,E1 -14637.679,E2 -14637.679} C_VEL
LIN {X 0,Y 337.475,Z 407.611,A -85,B 0,C 180,E1 -14638.8,E2 -14638.8} C_VEL
LIN {X 0,Y 336.507,Z 414.643,A -85,B 0,C 180,E1 -14639.918,E2 -14639.918} C_VEL
LIN {X 0,Y 335.758,Z 419.73,A -85,B 0,C 180,E1 -14640.879,E2 -14640.879} C_VEL
LIN {X 0,Y 334.995,Z 425.103,A -85,B 0,C 180,E1 -14642.094,E2 -14642.094} C_VEL
LIN {X 0,Y 334.26,Z 430.052,A -85,B 0,C 180,E1 -14643.462,E2 -14643.462} C_VEL
LIN {X 0,Y 333.602,Z 434.29,A -85,B 0,C 180,E1 -14644.929,E2 -14644.929} C_VEL
LIN {X 0,Y 333.048,Z 437.522,A -85,B 0,C 180,E1 -14646.363,E2 -14646.363} C_VEL
LIN {X 0,Y 332.499,Z 440.753,A -85,B 0,C 180,E1 -14648.422,E2 -14648.422} C_VEL
LIN {X 0,Y 332.134,Z 442.366,A -85,B 0,C 180,E1 -14650.211,E2 -14650.211} C_VEL
LIN {X 0,Y 331.969,Z 442.807,A -85,B 0,C 180,E1 -14652.284,E2 -14652.284} C_VEL
LIN {X 0,Y 331.924,Z 442.06,A -85,B 0,C 180,E1 -14654.023,E2 -14654.023} C_VEL
LIN {X 0,Y 332.024,Z 440.926,A -85,B 0,C 180,E1 -14655.286,E2 -14655.286} C_VEL
LIN {X 0,Y 332.178,Z 438.978,A -85,B 0,C 180,E1 -14656.689,E2 -14656.689} C_VEL
LIN {X 0,Y 332.456,Z 435.482,A -85,B 0,C 180,E1 -14658.415,E2 -14658.415} C_VEL
LIN {X 0,Y 332.669,Z 432.266,A -85,B 0,C 180,E1 -14659.655,E2 -14659.655} C_VEL
LIN {X 0,Y 333.091,Z 427.133,A -85,B 0,C 180,E1 -14661.201,E2 -14661.201} C_VEL
LIN {X 0,Y 333.423,Z 422.119,A -85,B 0,C 180,E1 -14662.435,E2 -14662.435} C_VEL
LIN {X 0,Y 333.948,Z 416.081,A -85,B 0,C 180,E1 -14663.657,E2 -14663.657} C_VEL
LIN {X 0,Y 334.535,Z 408.706,A -85,B 0,C 180,E1 -14664.878,E2 -14664.878} C_VEL
LIN {X 0,Y 335.061,Z 402.057,A -85,B 0,C 180,E1 -14665.79,E2 -14665.79} C_VEL
LIN {X 0,Y 335.627,Z 394.001,A -85,B 0,C 180,E1 -14666.699,E2 -14666.699} C_VEL
LIN {X 0,Y 336.143,Z 385.661,A -85,B 0,C 180,E1 -14667.454,E2 -14667.454} C_VEL
LIN {X 0,Y 336.509,Z 377.224,A -85,B 0,C 180,E1 -14668.055,E2 -14668.055} C_VEL
LIN {X 0,Y 336.853,Z 368.031,A -85,B 0,C 180,E1 -14668.543,E2 -14668.543} C_VEL
LIN {X 0,Y 337.084,Z 358.626,A -85,B 0,C 180,E1 -14668.879,E2 -14668.879} C_VEL
LIN {X 0,Y 337.868,Z 304.279,A -85,B 0,C 180,E1 -14670.055,E2 -14670.055} C_VEL
LIN {X 0,Y 334.506,Z 283.425,A -85,B 0,C 180,E1 -14670.666,E2 -14670.666} C_VEL
LIN {X 0,Y 334.086,Z 278.679,A -85,B 0,C 180,E1 -14672.185,E2 -14672.185} C_VEL
LIN {X 0,Y 333.98,Z 278.692,A -85,B 0,C 180,E1 -14676.04,E2 -14676.04} C_VEL
LIN {X 0,Y 333.925,Z 278.699,A -85,B 0,C 180,E1 -14678.472,E2 -14678.472} C_VEL
LIN {X 0,Y 333.757,Z 278.72,A -85,B 0,C 180,E1 -14682.156,E2 -14682.156} C_VEL
LIN {X 0,Y 333.776,Z 278.718,A -85,B 0,C 180,E1 -14684.636,E2 -14684.636} C_VEL
LIN {X 0,Y 333.764,Z 278.719,A -85,B 0,C 180,E1 -14688.657,E2 -14688.657} C_VEL
LIN {X 0,Y 333.66,Z 278.732,A -85,B 0,C 180,E1 -14692.281,E2 -14692.281} C_VEL
LIN {X 0,Y 333.659,Z 278.735,A -85,B 0,C 180,E1 -14695.092,E2 -14695.092} C_VEL
LIN {X 0,Y 333.624,Z 278.738,A -85,B 0,C 180,E1 -14698.981,E2 -14698.981} C_VEL
LIN {X 0,Y 333.616,Z 278.737,A -85,B 0,C 180,E1 -14702.59,E2 -14702.59} C_VEL
LIN {X 0,Y 333.649,Z 278.734,A -85,B 0,C 180,E1 -14706.143,E2 -14706.143} C_VEL
LIN {X 0,Y 333.581,Z 278.742,A -85,B 0,C 180,E1 -14709.016,E2 -14709.016} C_VEL
LIN {X 0,Y 332.896,Z 278.833,A -85,B 0,C 180,E1 -14710.024,E2 -14710.024} C_VEL
LIN {X 0,Y 330.031,Z 279.19,A -85,B 0,C 180,E1 -14711.663,E2 -14711.663} C_VEL
LIN {X 0,Y 327.615,Z 279.487,A -85,B 0,C 180,E1 -14712.991,E2 -14712.991} C_VEL
LIN {X 0,Y 326.582,Z 279.616,A -85,B 0,C 180,E1 -14714.019,E2 -14714.019} C_VEL
LIN {X 0,Y 326.5,Z 279.623,A -85,B 0,C 180,E1 -14714.367,E2 -14714.367} C_VEL
LIN {X 0,Y 326.557,Z 279.619,A -85,B 0,C 180,E1 -14718.158,E2 -14718.158} C_VEL
LIN {X 0,Y 326.605,Z 279.613,A -85,B 0,C 180,E1 -14721.396,E2 -14721.396} C_VEL
LIN {X 0,Y 326.603,Z 279.611,A -85,B 0,C 180,E1 -14724.856,E2 -14724.856} C_VEL
LIN {X 0,Y 326.594,Z 279.614,A -85,B 0,C 180,E1 -14727.46,E2 -14727.46} C_VEL
LIN {X 0,Y 326.603,Z 279.613,A -85,B 0,C 180,E1 -14730.341,E2 -14730.341} C_VEL
LIN {X 0,Y 326.632,Z 279.608,A -85,B 0,C 180,E1 -14734.649,E2 -14734.649} C_VEL
LIN {X 0,Y 326.613,Z 279.611,A -85,B 0,C 180,E1 -14738.548,E2 -14738.548} C_VEL
LIN {X 0,Y 326.848,Z 279.668,A -85,B 0,C 180,E1 -14742.566,E2 -14742.566} C_VEL
LIN {X 0,Y 326.813,Z 282.314,A -85,B 0,C 180,E1 -14743.289,E2 -14743.289} C_VEL
LIN {X 0,Y 328.976,Z 300.141,A -85,B 0,C 180,E1 -14743.92,E2 -14743.92} C_VEL
LIN {X 0,Y 329.367,Z 305.358,A -85,B 0,C 180,E1 -14744.09,E2 -14744.09} C_VEL
LIN {X 0,Y 328.126,Z 361.822,A -85,B 0,C 180,E1 -14745.864,E2 -14745.864} C_VEL
LIN {X 0,Y 327.875,Z 372.013,A -85,B 0,C 180,E1 -14746.367,E2 -14746.367} C_VEL
LIN {X 0,Y 327.461,Z 383.37,A -85,B 0,C 180,E1 -14747.139,E2 -14747.139} C_VEL
LIN {X 0,Y 327.116,Z 393.45,A -85,B 0,C 180,E1 -14748.07,E2 -14748.07} C_VEL
LIN {X 0,Y 326.629,Z 402.725,A -85,B 0,C 180,E1 -14749.153,E2 -14749.153} C_VEL
LIN {X 0,Y 326.165,Z 411.348,A -85,B 0,C 180,E1 -14750.391,E2 -14750.391} C_VEL
LIN {X 0,Y 325.763,Z 419.865,A -85,B 0,C 180,E1 -14751.943,E2 -14751.943} C_VEL
LIN {X 0,Y 325.463,Z 425.619,A -85,B 0,C 180,E1 -14753.246,E2 -14753.246} C_VEL
LIN {X 0,Y 325.276,Z 430.98,A -85,B 0,C 180,E1 -14754.735,E2 -14754.735} C_VEL
LIN {X 0,Y 325.148,Z 435.405,A -85,B 0,C 180,E1 -14756.286,E2 -14756.286} C_VEL
LIN {X 0,Y 324.949,Z 439.386,A -85,B 0,C 180,E1 -14758.145,E2 -14758.145} C_VEL
LIN {X 0,Y 324.977,Z 441.9,A -85,B 0,C 180,E1 -14760.004,E2 -14760.004} C_VEL
LIN {X 0,Y 325.065,Z 442.95,A -85,B 0,C 180,E1 -14761.243,E2 -14761.243} C_VEL
LIN {X 0,Y 325.253,Z 443.406,A -85,B 0,C 180,E1 -14762.481,E2 -14762.481} C_VEL
LIN {X 0,Y 325.575,Z 443.264,A -85,B 0,C 180,E1 -14763.717,E2 -14763.717} C_VEL
LIN {X 0,Y 325.946,Z 442.6,A -85,B 0,C 180,E1 -14764.952,E2 -14764.952} C_VEL
LIN {X 0,Y 326.229,Z 441.437,A -85,B 0,C 180,E1 -14766.187,E2 -14766.187} C_VEL
LIN {X 0,Y 326.429,Z 439.762,A -85,B 0,C 180,E1 -14767.426,E2 -14767.426} C_VEL
LIN {X 0,Y 327.268,Z 437.44,A -85,B 0,C 180,E1 -14768.649,E2 -14768.649} C_VEL
LIN {X 0,Y 327.809,Z 434.504,A -85,B 0,C 180,E1 -14769.88,E2 -14769.88} C_VEL
LIN {X 0,Y 329.142,Z 428.661,A -85,B 0,C 180,E1 -14771.707,E2 -14771.707} C_VEL
LIN {X 0,Y 330.37,Z 422.461,A -85,B 0,C 180,E1 -14773.223,E2 -14773.223} C_VEL
LIN {X 0,Y 331.833,Z 414.804,A -85,B 0,C 180,E1 -14774.727,E2 -14774.727} C_VEL
LIN {X 0,Y 333.305,Z 405.967,A -85,B 0,C 180,E1 -14776.07,E2 -14776.07} C_VEL
LIN {X 0,Y 334.499,Z 397.508,A -85,B 0,C 180,E1 -14777.11,E2 -14777.11} C_VEL
LIN {X 0,Y 335.839,Z 386.952,A -85,B 0,C 180,E1 -14778.14,E2 -14778.14} C_VEL
LIN {X 0,Y 336.935,Z 375.755,A -85,B 0,C 180,E1 -14778.945,E2 -14778.945} C_VEL
LIN {X 0,Y 337.715,Z 365.728,A -85,B 0,C 180,E1 -14779.484,E2 -14779.484} C_VEL
LIN {X 0,Y 341.102,Z 312.173,A -85,B 0,C 180,E1 -14781.398,E2 -14781.398} C_VEL
LIN {X 0,Y 339.868,Z 307.771,A -85,B 0,C 180,E1 -14781.758,E2 -14781.758} C_VEL
LIN {X 0,Y 335.313,Z 298.247,A -85,B 0,C 180,E1 -14782.862,E2 -14782.862} C_VEL
LIN {X 0,Y 330.573,Z 289.886,A -85,B 0,C 180,E1 -14784.039,E2 -14784.039} C_VEL
LIN {X 0,Y 328.87,Z 286.707,A -85,B 0,C 180,E1 -14784.528,E2 -14784.528} C_VEL
LIN {X 0,Y 326.621,Z 279.614,A -85,B 0,C 180,E1 -14787.473,E2 -14787.473} C_VEL
LIN {X 0,Y 326.583,Z 279.619,A -85,B 0,C 180,E1 -14791.099,E2 -14791.099} C_VEL
LIN {X 0,Y 326.616,Z 279.613,A -85,B 0,C 180,E1 -14794.022,E2 -14794.022} C_VEL
LIN {X 0,Y 326.632,Z 279.612,A -85,B 0,C 180,E1 -14797.239,E2 -14797.239} C_VEL
LIN {X 0,Y 326.555,Z 279.621,A -85,B 0,C 180,E1 -14801.126,E2 -14801.126} C_VEL
LIN {X 0,Y 326.571,Z 279.616,A -85,B 0,C 180,E1 -14803.527,E2 -14803.527} C_VEL
LIN {X 0,Y 326.586,Z 279.614,A -85,B 0,C 180,E1 -14807.03,E2 -14807.03} C_VEL
LIN {X 0,Y 326.609,Z 279.615,A -85,B 0,C 180,E1 -14810.777,E2 -14810.777} C_VEL
LIN {X 0,Y 326.622,Z 279.611,A -85,B 0,C 180,E1 -14814.481,E2 -14814.481} C_VEL
LIN {X 0,Y 326.618,Z 279.613,A -85,B 0,C 180,E1 -14817.456,E2 -14817.456} C_VEL
LIN {X 0,Y 326.658,Z 279.605,A -85,B 0,C 180,E1 -14820.34,E2 -14820.34} C_VEL
LIN {X 0,Y 326.713,Z 279.651,A -85,B 0,C 180,E1 -14822.315,E2 -14822.315} C_VEL
LIN {X 0,Y 329.407,Z 287.89,A -85,B 0,C 180,E1 -14824.092,E2 -14824.092} C_VEL
LIN {X 0,Y 331.384,Z 296.185,A -85,B 0,C 180,E1 -14825.504,E2 -14825.504} C_VEL
LIN {X 0,Y 331.863,Z 300.742,A -85,B 0,C 180,E1 -14826.065,E2 -14826.065} C_VEL
LIN {X 0,Y 334.771,Z 313.864,A -85,B 0,C 180,E1 -14827.145,E2 -14827.145} C_VEL
LIN {X 0,Y 337.43,Z 331.67,A -85,B 0,C 180,E1 -14828.343,E2 -14828.343} C_VEL
LIN {X 0,Y 338.748,Z 345.591,A -85,B 0,C 180,E1 -14829.135,E2 -14829.135} C_VEL
LIN {X 0,Y 338.788,Z 352.672,A -85,B 0,C 180,E1 -14829.452,E2 -14829.452} C_VEL
LIN {X 0,Y 336.344,Z 392.141,A -85,B 0,C 180,E1 -14830.865,E2 -14830.865} C_VEL
LIN {X 0,Y 335.04,Z 403.915,A -85,B 0,C 180,E1 -14831.502,E2 -14831.502} C_VEL
LIN {X 0,Y 333.737,Z 413.601,A -85,B 0,C 180,E1 -14832.221,E2 -14832.221} C_VEL
LIN {X 0,Y 332.179,Z 424.245,A -85,B 0,C 180,E1 -14833.245,E2 -14833.245} C_VEL
LIN {X 0,Y 330.661,Z 433.714,A -85,B 0,C 180,E1 -14834.434,E2 -14834.434} C_VEL
LIN {X 0,Y 329.509,Z 440.545,A -85,B 0,C 180,E1 -14835.486,E2 -14835.486} C_VEL
LIN {X 0,Y 328.412,Z 447.068,A -85,B 0,C 180,E1 -14836.7,E2 -14836.7} C_VEL
LIN {X 0,Y 327.442,Z 452.531,A -85,B 0,C 180,E1 -14837.92,E2 -14837.92} C_VEL
LIN {X 0,Y 326.541,Z 458.137,A -85,B 0,C 180,E1 -14839.459,E2 -14839.459} C_VEL
LIN {X 0,Y 325.706,Z 463.421,A -85,B 0,C 180,E1 -14841.312,E2 -14841.312} C_VEL
LIN {X 0,Y 325.181,Z 467.117,A -85,B 0,C 180,E1 -14843.173,E2 -14843.173} C_VEL
LIN {X 0,Y 324.963,Z 469.501,A -85,B 0,C 180,E1 -14845.037,E2 -14845.037} C_VEL
LIN {X 0,Y 324.983,Z 470.443,A -85,B 0,C 180,E1 -14846.28,E2 -14846.28} C_VEL
LIN {X 0,Y 324.945,Z 470.881,A -85,B 0,C 180,E1 -14847.521,E2 -14847.521} C_VEL
LIN {X 0,Y 325.015,Z 472.055,A -85,B 0,C 180,E1 -14848.761,E2 -14848.761} C_VEL
LIN {X 0,Y 325.044,Z 472.776,A -85,B 0,C 180,E1 -14850,E2 -14850} C_VEL
LIN {X 0,Y 324.95,Z 473.016,A -85,B 0,C 180,E1 -14851.239,E2 -14851.239} C_VEL
LIN {X 0,Y 324.906,Z 472.671,A -85,B 0,C 180,E1 -14852.479,E2 -14852.479} C_VEL
LIN {X 0,Y 324.968,Z 471.818,A -85,B 0,C 180,E1 -14853.72,E2 -14853.72} C_VEL
LIN {X 0,Y 325.011,Z 469.244,A -85,B 0,C 180,E1 -14855.884,E2 -14855.884} C_VEL
LIN {X 0,Y 325.308,Z 466.308,A -85,B 0,C 180,E1 -14857.448,E2 -14857.448} C_VEL
LIN {X 0,Y 325.847,Z 461.493,A -85,B 0,C 180,E1 -14859.309,E2 -14859.309} C_VEL
LIN {X 0,Y 326.555,Z 456.317,A -85,B 0,C 180,E1 -14860.854,E2 -14860.854} C_VEL
LIN {X 0,Y 327.301,Z 451.274,A -85,B 0,C 180,E1 -14862.084,E2 -14862.084} C_VEL
LIN {X 0,Y 328.167,Z 445.22,A -85,B 0,C 180,E1 -14863.31,E2 -14863.31} C_VEL
LIN {X 0,Y 329.194,Z 437.875,A -85,B 0,C 180,E1 -14864.528,E2 -14864.528} C_VEL
LIN {X 0,Y 330.283,Z 430.027,A -85,B 0,C 180,E1 -14865.583,E2 -14865.583} C_VEL
LIN {X 0,Y 331.363,Z 421.755,A -85,B 0,C 180,E1 -14866.479,E2 -14866.479} C_VEL
LIN {X 0,Y 332.417,Z 411.261,A -85,B 0,C 180,E1 -14867.375,E2 -14867.375} C_VEL
LIN {X 0,Y 333.417,Z 400.005,A -85,B 0,C 180,E1 -14868.034,E2 -14868.034} C_VEL
LIN {X 0,Y 333.967,Z 389.784,A -85,B 0,C 180,E1 -14868.434,E2 -14868.434} C_VEL
LIN {X 0,Y 334.873,Z 348.587,A -85,B 0,C 180,E1 -14869.366,E2 -14869.366} C_VEL
LIN {X 0,Y 332.493,Z 331.27,A -85,B 0,C 180,E1 -14869.95,E2 -14869.95} C_VEL
LIN {X 0,Y 328.644,Z 311.365,A -85,B 0,C 180,E1 -14870.748,E2 -14870.748} C_VEL
LIN {X 0,Y 330.157,Z 297.85,A -85,B 0,C 180,E1 -14874.525,E2 -14874.525} C_VEL
LIN {X 0,Y 328.662,Z 288.667,A -85,B 0,C 180,E1 -14877.371,E2 -14877.371} C_VEL
LIN {X 0,Y 326.638,Z 279.608,A -85,B 0,C 180,E1 -14880.378,E2 -14880.378} C_VEL
LIN {X 0,Y 326.615,Z 279.616,A -85,B 0,C 180,E1 -14884.018,E2 -14884.018} C_VEL
LIN {X 0,Y 326.631,Z 279.609,A -85,B 0,C 180,E1 -14887.235,E2 -14887.235} C_VEL
LIN {X 0,Y 326.584,Z 279.615,A -85,B 0,C 180,E1 -14891.129,E2 -14891.129} C_VEL
LIN {X 0,Y 326.535,Z 279.618,A -85,B 0,C 180,E1 -14894.741,E2 -14894.741} C_VEL
LIN {X 0,Y 326.571,Z 279.617,A -85,B 0,C 180,E1 -14898.15,E2 -14898.15} C_VEL
LIN {X 0,Y 326.575,Z 279.612,A -85,B 0,C 180,E1 -14901.381,E2 -14901.381} C_VEL
LIN {X 0,Y 326.627,Z 279.603,A -85,B 0,C 180,E1 -14904.849,E2 -14904.849} C_VEL
LIN {X 0,Y 326.615,Z 279.614,A -85,B 0,C 180,E1 -14907.453,E2 -14907.453} C_VEL
LIN {X 0,Y 326.623,Z 279.61,A -85,B 0,C 180,E1 -14910.334,E2 -14910.334} C_VEL
LIN {X 0,Y 326.624,Z 279.606,A -85,B 0,C 180,E1 -14913.134,E2 -14913.134} C_VEL
LIN {X 0,Y 326.647,Z 279.611,A -85,B 0,C 180,E1 -14915.867,E2 -14915.867} C_VEL
LIN {X 0,Y 326.636,Z 279.605,A -85,B 0,C 180,E1 -14919.86,E2 -14919.86} C_VEL
LIN {X 0,Y 326.669,Z 279.599,A -85,B 0,C 180,E1 -14922.467,E2 -14922.467} C_VEL
LIN {X 0,Y 326.764,Z 279.591,A -85,B 0,C 180,E1 -14926.311,E2 -14926.311} C_VEL
LIN {X 0,Y 326.809,Z 279.579,A -85,B 0,C 180,E1 -14930.09,E2 -14930.09} C_VEL
LIN {X 0,Y 326.99,Z 279.555,A -85,B 0,C 180,E1 -14933.827,E2 -14933.827} C_VEL
LIN {X 0,Y 327.035,Z 279.555,A -85,B 0,C 180,E1 -14937.533,E2 -14937.533} C_VEL
LIN {X 0,Y 327.158,Z 279.532,A -85,B 0,C 180,E1 -14939.996,E2 -14939.996} C_VEL
LIN {X 0,Y 327.041,Z 279.557,A -85,B 0,C 180,E1 -14942.459,E2 -14942.459} C_VEL
LIN {X 0,Y 326.926,Z 279.564,A -85,B 0,C 180,E1 -14946.505,E2 -14946.505} C_VEL
LIN {X 0,Y 326.779,Z 279.586,A -85,B 0,C 180,E1 -14949.903,E2 -14949.903} C_VEL
LIN {X 0,Y 326.753,Z 279.595,A -85,B 0,C 180,E1 -14953.681,E2 -14953.681} C_VEL
LIN {X 0,Y 326.691,Z 279.6,A -85,B 0,C 180,E1 -14957.523,E2 -14957.523} C_VEL
LIN {X 0,Y 326.654,Z 279.602,A -85,B 0,C 180,E1 -14960.131,E2 -14960.131} C_VEL
LIN {X 0,Y 326.641,Z 279.606,A -85,B 0,C 180,E1 -14964.124,E2 -14964.124} C_VEL
LIN {X 0,Y 326.67,Z 279.606,A -85,B 0,C 180,E1 -14966.853,E2 -14966.853} C_VEL
LIN {X 0,Y 326.619,Z 279.613,A -85,B 0,C 180,E1 -14970.605,E2 -14970.605} C_VEL
LIN {X 0,Y 326.59,Z 279.616,A -85,B 0,C 180,E1 -14974.015,E2 -14974.015} C_VEL
LIN {X 0,Y 326.609,Z 279.61,A -85,B 0,C 180,E1 -14977.234,E2 -14977.234} C_VEL
LIN {X 0,Y 326.614,Z 279.605,A -85,B 0,C 180,E1 -14980.199,E2 -14980.199} C_VEL
LIN {X 0,Y 326.636,Z 279.607,A -85,B 0,C 180,E1 -14983.506,E2 -14983.506} C_VEL
LIN {X 0,Y 326.626,Z 279.608,A -85,B 0,C 180,E1 -14987.011,E2 -14987.011} C_VEL
LIN {X 0,Y 326.672,Z 279.74,A -85,B 0,C 180,E1 -14990.599,E2 -14990.599} C_VEL
LIN {X 0,Y 327.649,Z 284.312,A -85,B 0,C 180,E1 -14992.194,E2 -14992.194} C_VEL
LIN {X 0,Y 333.76,Z 299.513,A -85,B 0,C 180,E1 -14993.077,E2 -14993.077} C_VEL
LIN {X 0,Y 335.68,Z 308.207,A -85,B 0,C 180,E1 -14993.432,E2 -14993.432} C_VEL
LIN {X 0,Y 334.488,Z 360.719,A -85,B 0,C 180,E1 -14994.603,E2 -14994.603} C_VEL
LIN {X 0,Y 334.132,Z 370.161,A -85,B 0,C 180,E1 -14994.969,E2 -14994.969} C_VEL
LIN {X 0,Y 333.508,Z 381.043,A -85,B 0,C 180,E1 -14995.597,E2 -14995.597} C_VEL
LIN {X 0,Y 332.508,Z 391.872,A -85,B 0,C 180,E1 -14996.483,E2 -14996.483} C_VEL
LIN {X 0,Y 331.625,Z 400.888,A -85,B 0,C 180,E1 -14997.469,E2 -14997.469} C_VEL
LIN {X 0,Y 330.704,Z 408.253,A -85,B 0,C 180,E1 -14998.458,E2 -14998.458} C_VEL
LIN {X 0,Y 329.696,Z 415.165,A -85,B 0,C 180,E1 -14999.585,E2 -14999.585} C_VEL
LIN {X 0,Y 328.753,Z 421.255,A -85,B 0,C 180,E1 -15000.791,E2 -15000.791} C_VEL
LIN {X 0,Y 328.055,Z 425.857,A -85,B 0,C 180,E1 -15001.881,E2 -15001.881} C_VEL
LIN {X 0,Y 327.333,Z 430.49,A -85,B 0,C 180,E1 -15003.2,E2 -15003.2} C_VEL
LIN {X 0,Y 326.645,Z 434.545,A -85,B 0,C 180,E1 -15004.63,E2 -15004.63} C_VEL
LIN {X 0,Y 325.928,Z 438.518,A -85,B 0,C 180,E1 -15006.49,E2 -15006.49} C_VEL
LIN {X 0,Y 325.482,Z 441.023,A -85,B 0,C 180,E1 -15008.183,E2 -15008.183} C_VEL
LIN {X 0,Y 325.108,Z 442.476,A -85,B 0,C 180,E1 -15009.765,E2 -15009.765} C_VEL
LIN {X 0,Y 324.889,Z 443.153,A -85,B 0,C 180,E1 -15012.12,E2 -15012.12} C_VEL
LIN {X 0,Y 324.845,Z 442.618,A -85,B 0,C 180,E1 -15013.665,E2 -15013.665} C_VEL
LIN {X 0,Y 324.908,Z 441.588,A -85,B 0,C 180,E1 -15014.956,E2 -15014.956} C_VEL
LIN {X 0,Y 325.079,Z 439.445,A -85,B 0,C 180,E1 -15016.597,E2 -15016.597} C_VEL
LIN {X 0,Y 325.311,Z 436.505,A -85,B 0,C 180,E1 -15018.157,E2 -15018.157} C_VEL
LIN {X 0,Y 325.691,Z 431.515,A -85,B 0,C 180,E1 -15020.059,E2 -15020.059} C_VEL
LIN {X 0,Y 326.05,Z 427.339,A -85,B 0,C 180,E1 -15021.322,E2 -15021.322} C_VEL
LIN {X 0,Y 326.374,Z 422.326,A -85,B 0,C 180,E1 -15022.577,E2 -15022.577} C_VEL
LIN {X 0,Y 326.92,Z 416.235,A -85,B 0,C 180,E1 -15023.83,E2 -15023.83} C_VEL
LIN {X 0,Y 327.524,Z 408.825,A -85,B 0,C 180,E1 -15025.076,E2 -15025.076} C_VEL
LIN {X 0,Y 328.08,Z 402.129,A -85,B 0,C 180,E1 -15026.008,E2 -15026.008} C_VEL
LIN {X 0,Y 328.658,Z 394.017,A -85,B 0,C 180,E1 -15026.936,E2 -15026.936} C_VEL
LIN {X 0,Y 329.19,Z 385.599,A -85,B 0,C 180,E1 -15027.706,E2 -15027.706} C_VEL
LIN {X 0,Y 329.587,Z 377.037,A -85,B 0,C 180,E1 -15028.32,E2 -15028.32} C_VEL
LIN {X 0,Y 329.961,Z 366.979,A -85,B 0,C 180,E1 -15028.849,E2 -15028.849} C_VEL
LIN {X 0,Y 330.216,Z 355.587,A -85,B 0,C 180,E1 -15029.225,E2 -15029.225} C_VEL
LIN {X 0,Y 330.919,Z 304.88,A -85,B 0,C 180,E1 -15030.324,E2 -15030.324} C_VEL
LIN {X 0,Y 327.484,Z 283.672,A -85,B 0,C 180,E1 -15030.98,E2 -15030.98} C_VEL
LIN {X 0,Y 327.046,Z 279.556,A -85,B 0,C 180,E1 -15032.309,E2 -15032.309} C_VEL
LIN {X 0,Y 326.955,Z 279.567,A -85,B 0,C 180,E1 -15036.17,E2 -15036.17} C_VEL
LIN {X 0,Y 326.772,Z 279.591,A -85,B 0,C 180,E1 -15039.908,E2 -15039.908} C_VEL
LIN {X 0,Y 326.723,Z 279.598,A -85,B 0,C 180,E1 -15043.687,E2 -15043.687} C_VEL
LIN {X 0,Y 326.667,Z 279.607,A -85,B 0,C 180,E1 -15047.53,E2 -15047.53} C_VEL
LIN {X 0,Y 326.634,Z 279.607,A -85,B 0,C 180,E1 -15050.137,E2 -15050.137} C_VEL
LIN {X 0,Y 326.603,Z 279.611,A -85,B 0,C 180,E1 -15054.133,E2 -15054.133} C_VEL
LIN {X 0,Y 326.57,Z 279.615,A -85,B 0,C 180,E1 -15058.259,E2 -15058.259} C_VEL
LIN {X 0,Y 326.545,Z 279.62,A -85,B 0,C 180,E1 -15061.1,E2 -15061.1} C_VEL
LIN {X 0,Y 326.58,Z 279.616,A -85,B 0,C 180,E1 -15064.023,E2 -15064.023} C_VEL
LIN {X 0,Y 326.597,Z 279.614,A -85,B 0,C 180,E1 -15067.241,E2 -15067.241} C_VEL
LIN {X 0,Y 326.521,Z 279.622,A -85,B 0,C 180,E1 -15071.128,E2 -15071.128} C_VEL
LIN {X 0,Y 326.5,Z 279.623,A -85,B 0,C 180,E1 -15074.367,E2 -15074.367} C_VEL
LIN {X 0,Y 325.832,Z 279.712,A -85,B 0,C 180,E1 -15075.397,E2 -15075.397} C_VEL
LIN {X 0,Y 322.973,Z 280.064,A -85,B 0,C 180,E1 -15077.072,E2 -15077.072} C_VEL
LIN {X 0,Y 320.57,Z 280.363,A -85,B 0,C 180,E1 -15078.429,E2 -15078.429} C_VEL
LIN {X 0,Y 319.569,Z 280.49,A -85,B 0,C 180,E1 -15079.481,E2 -15079.481} C_VEL
LIN {X 0,Y 319.504,Z 280.493,A -85,B 0,C 180,E1 -15079.836,E2 -15079.836} C_VEL
LIN {X 0,Y 319.542,Z 280.494,A -85,B 0,C 180,E1 -15083.577,E2 -15083.577} C_VEL
LIN {X 0,Y 319.563,Z 280.488,A -85,B 0,C 180,E1 -15086.691,E2 -15086.691} C_VEL
LIN {X 0,Y 319.547,Z 280.493,A -85,B 0,C 180,E1 -15089.618,E2 -15089.618} C_VEL
LIN {X 0,Y 319.534,Z 280.493,A -85,B 0,C 180,E1 -15092.497,E2 -15092.497} C_VEL
LIN {X 0,Y 319.564,Z 280.488,A -85,B 0,C 180,E1 -15095.306,E2 -15095.306} C_VEL
LIN {X 0,Y 319.597,Z 280.483,A -85,B 0,C 180,E1 -15099.405,E2 -15099.405} C_VEL
LIN {X 0,Y 319.783,Z 280.545,A -85,B 0,C 180,E1 -15102.581,E2 -15102.581} C_VEL
LIN {X 0,Y 319.793,Z 282.861,A -85,B 0,C 180,E1 -15103.158,E2 -15103.158} C_VEL
LIN {X 0,Y 322.113,Z 302.097,A -85,B 0,C 180,E1 -15103.835,E2 -15103.835} C_VEL
LIN {X 0,Y 322.254,Z 307.36,A -85,B 0,C 180,E1 -15104.007,E2 -15104.007} C_VEL
LIN {X 0,Y 321.051,Z 362.176,A -85,B 0,C 180,E1 -15105.788,E2 -15105.788} C_VEL
LIN {X 0,Y 320.788,Z 372.261,A -85,B 0,C 180,E1 -15106.302,E2 -15106.302} C_VEL
LIN {X 0,Y 320.368,Z 383.557,A -85,B 0,C 180,E1 -15107.091,E2 -15107.091} C_VEL
LIN {X 0,Y 320.033,Z 394.365,A -85,B 0,C 180,E1 -15108.124,E2 -15108.124} C_VEL
LIN {X 0,Y 319.454,Z 403.484,A -85,B 0,C 180,E1 -15109.227,E2 -15109.227} C_VEL
LIN {X 0,Y 319.047,Z 412.027,A -85,B 0,C 180,E1 -15110.495,E2 -15110.495} C_VEL
LIN {X 0,Y 318.664,Z 420.439,A -85,B 0,C 180,E1 -15112.081,E2 -15112.081} C_VEL
LIN {X 0,Y 318.274,Z 427.135,A -85,B 0,C 180,E1 -15113.665,E2 -15113.665} C_VEL
LIN {X 0,Y 318.158,Z 433.477,A -85,B 0,C 180,E1 -15115.57,E2 -15115.57} C_VEL
LIN {X 0,Y 317.911,Z 438.015,A -85,B 0,C 180,E1 -15117.47,E2 -15117.47} C_VEL
LIN {X 0,Y 317.854,Z 440.315,A -85,B 0,C 180,E1 -15118.737,E2 -15118.737} C_VEL
LIN {X 0,Y 317.881,Z 442.043,A -85,B 0,C 180,E1 -15120.004,E2 -15120.004} C_VEL
LIN {X 0,Y 317.97,Z 443.165,A -85,B 0,C 180,E1 -15121.271,E2 -15121.271} C_VEL
LIN {X 0,Y 318.166,Z 443.692,A -85,B 0,C 180,E1 -15122.536,E2 -15122.536} C_VEL
LIN {X 0,Y 318.503,Z 443.693,A -85,B 0,C 180,E1 -15123.8,E2 -15123.8} C_VEL
LIN {X 0,Y 318.891,Z 443.18,A -85,B 0,C 180,E1 -15125.061,E2 -15125.061} C_VEL
LIN {X 0,Y 319.209,Z 442.16,A -85,B 0,C 180,E1 -15126.324,E2 -15126.324} C_VEL
LIN {X 0,Y 319.443,Z 440.609,A -85,B 0,C 180,E1 -15127.589,E2 -15127.589} C_VEL
LIN {X 0,Y 320.556,Z 437.176,A -85,B 0,C 180,E1 -15129.389,E2 -15129.389} C_VEL
LIN {X 0,Y 321.821,Z 432.04,A -85,B 0,C 180,E1 -15131.339,E2 -15131.339} C_VEL
LIN {X 0,Y 323.334,Z 425.463,A -85,B 0,C 180,E1 -15133.196,E2 -15133.196} C_VEL
LIN {X 0,Y 324.829,Z 418.29,A -85,B 0,C 180,E1 -15134.731,E2 -15134.731} C_VEL
LIN {X 0,Y 326.162,Z 411.268,A -85,B 0,C 180,E1 -15135.95,E2 -15135.95} C_VEL
LIN {X 0,Y 327.824,Z 401.619,A -85,B 0,C 180,E1 -15137.308,E2 -15137.308} C_VEL
LIN {X 0,Y 329.207,Z 391.993,A -85,B 0,C 180,E1 -15138.357,E2 -15138.357} C_VEL
LIN {X 0,Y 330.259,Z 383.467,A -85,B 0,C 180,E1 -15139.101,E2 -15139.101} C_VEL
LIN {X 0,Y 331.34,Z 372.607,A -85,B 0,C 180,E1 -15139.842,E2 -15139.842} C_VEL
LIN {X 0,Y 332.32,Z 359.736,A -85,B 0,C 180,E1 -15140.426,E2 -15140.426} C_VEL
LIN {X 0,Y 335.521,Z 314.197,A -85,B 0,C 180,E1 -15142.069,E2 -15142.069} C_VEL
LIN {X 0,Y 334.437,Z 310.804,A -85,B 0,C 180,E1 -15142.386,E2 -15142.386} C_VEL
LIN {X 0,Y 330.262,Z 302.06,A -85,B 0,C 180,E1 -15143.454,E2 -15143.454} C_VEL
LIN {X 0,Y 325.532,Z 293.546,A -85,B 0,C 180,E1 -15144.712,E2 -15144.712} C_VEL
LIN {X 0,Y 321.822,Z 287.293,A -85,B 0,C 180,E1 -15145.824,E2 -15145.824} C_VEL
LIN {X 0,Y 319.564,Z 280.492,A -85,B 0,C 180,E1 -15148.856,E2 -15148.856} C_VEL
LIN {X 0,Y 319.534,Z 280.496,A -85,B 0,C 180,E1 -15151.865,E2 -15151.865} C_VEL
LIN {X 0,Y 319.588,Z 280.488,A -85,B 0,C 180,E1 -15155.544,E2 -15155.544} C_VEL
LIN {X 0,Y 319.539,Z 280.495,A -85,B 0,C 180,E1 -15159.664,E2 -15159.664} C_VEL
LIN {X 0,Y 319.531,Z 280.493,A -85,B 0,C 180,E1 -15163.462,E2 -15163.462} C_VEL
LIN {X 0,Y 319.564,Z 280.489,A -85,B 0,C 180,E1 -15167.018,E2 -15167.018} C_VEL
LIN {X 0,Y 319.556,Z 280.491,A -85,B 0,C 180,E1 -15170.372,E2 -15170.372} C_VEL
LIN {X 0,Y 319.59,Z 280.487,A -85,B 0,C 180,E1 -15174.459,E2 -15174.459} C_VEL
LIN {X 0,Y 319.541,Z 280.49,A -85,B 0,C 180,E1 -15178.139,E2 -15178.139} C_VEL
LIN {X 0,Y 319.614,Z 280.606,A -85,B 0,C 180,E1 -15180.798,E2 -15180.798} C_VEL
LIN {X 0,Y 320.297,Z 282.785,A -85,B 0,C 180,E1 -15181.369,E2 -15181.369} C_VEL
LIN {X 0,Y 321.78,Z 284.755,A -85,B 0,C 180,E1 -15182.062,E2 -15182.062} C_VEL
LIN {X 0,Y 324.226,Z 292.305,A -85,B 0,C 180,E1 -15183.721,E2 -15183.721} C_VEL
LIN {X 0,Y 325.936,Z 299.994,A -85,B 0,C 180,E1 -15185.034,E2 -15185.034} C_VEL
LIN {X 0,Y 329.056,Z 314.529,A -85,B 0,C 180,E1 -15186.323,E2 -15186.323} C_VEL
LIN {X 0,Y 331.072,Z 327.726,A -85,B 0,C 180,E1 -15187.28,E2 -15187.28} C_VEL
LIN {X 0,Y 332.688,Z 342.392,A -85,B 0,C 180,E1 -15188.217,E2 -15188.217} C_VEL
LIN {X 0,Y 333.069,Z 352.472,A -85,B 0,C 180,E1 -15188.728,E2 -15188.728} C_VEL
LIN {X 0,Y 330.389,Z 391.618,A -85,B 0,C 180,E1 -15190.182,E2 -15190.182} C_VEL
LIN {X 0,Y 329.023,Z 403.313,A -85,B 0,C 180,E1 -15190.827,E2 -15190.827} C_VEL
LIN {X 0,Y 327.663,Z 413.029,A -85,B 0,C 180,E1 -15191.556,E2 -15191.556} C_VEL
LIN {X 0,Y 326.002,Z 423.711,A -85,B 0,C 180,E1 -15192.595,E2 -15192.595} C_VEL
LIN {X 0,Y 324.34,Z 433.141,A -85,B 0,C 180,E1 -15193.8,E2 -15193.8} C_VEL
LIN {X 0,Y 323.082,Z 439.947,A -85,B 0,C 180,E1 -15194.868,E2 -15194.868} C_VEL
LIN {X 0,Y 321.57,Z 447.963,A -85,B 0,C 180,E1 -15196.411,E2 -15196.411} C_VEL
LIN {X 0,Y 320.324,Z 454.466,A -85,B 0,C 180,E1 -15197.969,E2 -15197.969} C_VEL
LIN {X 0,Y 319.244,Z 460.444,A -85,B 0,C 180,E1 -15199.856,E2 -15199.856} C_VEL
LIN {X 0,Y 318.463,Z 464.885,A -85,B 0,C 180,E1 -15201.752,E2 -15201.752} C_VEL
LIN {X 0,Y 317.989,Z 468.034,A -85,B 0,C 180,E1 -15203.655,E2 -15203.655} C_VEL
LIN {X 0,Y 317.878,Z 469.356,A -85,B 0,C 180,E1 -15204.926,E2 -15204.926} C_VEL
LIN {X 0,Y 317.887,Z 470.157,A -85,B 0,C 180,E1 -15206.197,E2 -15206.197} C_VEL
LIN {X 0,Y 317.862,Z 470.452,A -85,B 0,C 180,E1 -15207.465,E2 -15207.465} C_VEL
LIN {X 0,Y 317.919,Z 471.657,A -85,B 0,C 180,E1 -15208.733,E2 -15208.733} C_VEL
LIN {X 0,Y 317.952,Z 472.424,A -85,B 0,C 180,E1 -15210,E2 -15210} C_VEL
LIN {X 0,Y 317.855,Z 472.691,A -85,B 0,C 180,E1 -15211.267,E2 -15211.267} C_VEL
LIN {X 0,Y 317.825,Z 472.366,A -85,B 0,C 180,E1 -15212.535,E2 -15212.535} C_VEL
LIN {X 0,Y 317.873,Z 471.56,A -85,B 0,C 180,E1 -15213.803,E2 -15213.803} C_VEL
LIN {X 0,Y 317.917,Z 469.291,A -85,B 0,C 180,E1 -15215.833,E2 -15215.833} C_VEL
LIN {X 0,Y 318.247,Z 466.17,A -85,B 0,C 180,E1 -15217.614,E2 -15217.614} C_VEL
LIN {X 0,Y 318.845,Z 461.447,A -85,B 0,C 180,E1 -15219.515,E2 -15219.515} C_VEL
LIN {X 0,Y 319.587,Z 456.335,A -85,B 0,C 180,E1 -15221.094,E2 -15221.094} C_VEL
LIN {X 0,Y 320.364,Z 451.364,A -85,B 0,C 180,E1 -15222.35,E2 -15222.35} C_VEL
LIN {X 0,Y 321.246,Z 445.395,A -85,B 0,C 180,E1 -15223.602,E2 -15223.602} C_VEL
LIN {X 0,Y 322.358,Z 438.148,A -85,B 0,C 180,E1 -15224.843,E2 -15224.843} C_VEL
LIN {X 0,Y 323.482,Z 430.423,A -85,B 0,C 180,E1 -15225.92,E2 -15225.92} C_VEL
LIN {X 0,Y 324.401,Z 423.805,A -85,B 0,C 180,E1 -15226.682,E2 -15226.682} C_VEL
LIN {X 0,Y 325.282,Z 415.773,A -85,B 0,C 180,E1 -15227.444,E2 -15227.444} C_VEL
LIN {X 0,Y 326.169,Z 406.527,A -85,B 0,C 180,E1 -15228.124,E2 -15228.124} C_VEL
LIN {X 0,Y 326.978,Z 397.531,A -85,B 0,C 180,E1 -15228.605,E2 -15228.605} C_VEL
LIN {X 0,Y 327.525,Z 388.044,A -85,B 0,C 180,E1 -15228.952,E2 -15228.952} C_VEL
LIN {X 0,Y 328.259,Z 347.974,A -85,B 0,C 180,E1 -15229.881,E2 -15229.881} C_VEL
LIN {X 0,Y 325.55,Z 329.568,A -85,B 0,C 180,E1 -15230.54,E2 -15230.54} C_VEL
LIN {X 0,Y 321.843,Z 310.934,A -85,B 0,C 180,E1 -15231.34,E2 -15231.34} C_VEL
LIN {X 0,Y 323.241,Z 299.041,A -85,B 0,C 180,E1 -15234.742,E2 -15234.742} C_VEL
LIN {X 0,Y 321.721,Z 289.882,A -85,B 0,C 180,E1 -15237.659,E2 -15237.659} C_VEL
LIN {X 0,Y 319.568,Z 280.492,A -85,B 0,C 180,E1 -15240.876,E2 -15240.876} C_VEL
LIN {X 0,Y 319.586,Z 280.487,A -85,B 0,C 180,E1 -15243.351,E2 -15243.351} C_VEL
LIN {X 0,Y 319.564,Z 280.483,A -85,B 0,C 180,E1 -15246.427,E2 -15246.427} C_VEL
LIN {X 0,Y 319.568,Z 280.491,A -85,B 0,C 180,E1 -15249.667,E2 -15249.667} C_VEL
LIN {X 0,Y 319.53,Z 280.495,A -85,B 0,C 180,E1 -15253.459,E2 -15253.459} C_VEL
LIN {X 0,Y 319.561,Z 280.489,A -85,B 0,C 180,E1 -15257.014,E2 -15257.014} C_VEL
LIN {X 0,Y 319.523,Z 280.491,A -85,B 0,C 180,E1 -15260.364,E2 -15260.364} C_VEL
LIN {X 0,Y 319.587,Z 280.48,A -85,B 0,C 180,E1 -15264.455,E2 -15264.455} C_VEL
LIN {X 0,Y 319.531,Z 280.489,A -85,B 0,C 180,E1 -15268.135,E2 -15268.135} C_VEL
LIN {X 0,Y 319.595,Z 280.489,A -85,B 0,C 180,E1 -15271.595,E2 -15271.595} C_VEL
LIN {X 0,Y 319.587,Z 280.485,A -85,B 0,C 180,E1 -15275.299,E2 -15275.299} C_VEL
LIN {X 0,Y 319.573,Z 280.48,A -85,B 0,C 180,E1 -15278.043,E2 -15278.043} C_VEL
LIN {X 0,Y 319.63,Z 280.479,A -85,B 0,C 180,E1 -15282.068,E2 -15282.068} C_VEL
LIN {X 0,Y 319.737,Z 280.469,A -85,B 0,C 180,E1 -15286.004,E2 -15286.004} C_VEL
LIN {X 0,Y 319.756,Z 280.455,A -85,B 0,C 180,E1 -15289.869,E2 -15289.869} C_VEL
LIN {X 0,Y 319.915,Z 280.441,A -85,B 0,C 180,E1 -15292.422,E2 -15292.422} C_VEL
LIN {X 0,Y 319.738,Z 280.455,A -85,B 0,C 180,E1 -15294.952,E2 -15294.952} C_VEL
LIN {X 0,Y 319.978,Z 280.434,A -85,B 0,C 180,E1 -15297.478,E2 -15297.478} C_VEL
LIN {X 0,Y 320.111,Z 280.41,A -85,B 0,C 180,E1 -15299.996,E2 -15299.996} C_VEL
LIN {X 0,Y 319.985,Z 280.436,A -85,B 0,C 180,E1 -15302.514,E2 -15302.514} C_VEL
LIN {X 0,Y 319.891,Z 280.441,A -85,B 0,C 180,E1 -15306.49,E2 -15306.49} C_VEL
LIN {X 0,Y 319.731,Z 280.462,A -85,B 0,C 180,E1 -15310.124,E2 -15310.124} C_VEL
LIN {X 0,Y 319.726,Z 280.472,A -85,B 0,C 180,E1 -15313.988,E2 -15313.988} C_VEL
LIN {X 0,Y 319.65,Z 280.48,A -85,B 0,C 180,E1 -15317.922,E2 -15317.922} C_VEL
LIN {X 0,Y 319.605,Z 280.479,A -85,B 0,C 180,E1 -15320.594,E2 -15320.594} C_VEL
LIN {X 0,Y 319.559,Z 280.489,A -85,B 0,C 180,E1 -15323.315,E2 -15323.315} C_VEL
LIN {X 0,Y 319.622,Z 280.482,A -85,B 0,C 180,E1 -15326.084,E2 -15326.084} C_VEL
LIN {X 0,Y 319.566,Z 280.489,A -85,B 0,C 180,E1 -15328.93,E2 -15328.93} C_VEL
LIN {X 0,Y 319.514,Z 280.493,A -85,B 0,C 180,E1 -15331.858,E2 -15331.858} C_VEL
LIN {X 0,Y 319.562,Z 280.477,A -85,B 0,C 180,E1 -15335.539,E2 -15335.539} C_VEL
LIN {X 0,Y 319.563,Z 280.491,A -85,B 0,C 180,E1 -15338.003,E2 -15338.003} C_VEL
LIN {X 0,Y 319.58,Z 280.489,A -85,B 0,C 180,E1 -15341.608,E2 -15341.608} C_VEL
LIN {X 0,Y 319.623,Z 280.486,A -85,B 0,C 180,E1 -15345.281,E2 -15345.281} C_VEL
LIN {X 0,Y 319.559,Z 280.491,A -85,B 0,C 180,E1 -15348.717,E2 -15348.717} C_VEL
LIN {X 0,Y 319.62,Z 280.647,A -85,B 0,C 180,E1 -15350.138,E2 -15350.138} C_VEL
LIN {X 0,Y 320.517,Z 284.761,A -85,B 0,C 180,E1 -15351.609,E2 -15351.609} C_VEL
LIN {X 0,Y 327.685,Z 302.384,A -85,B 0,C 180,E1 -15352.654,E2 -15352.654} C_VEL
LIN {X 0,Y 329.158,Z 308.877,A -85,B 0,C 180,E1 -15352.931,E2 -15352.931} C_VEL
LIN {X 0,Y 327.949,Z 361.796,A -85,B 0,C 180,E1 -15354.146,E2 -15354.146} C_VEL
LIN {X 0,Y 327.505,Z 372.514,A -85,B 0,C 180,E1 -15354.592,E2 -15354.592} C_VEL
LIN {X 0,Y 326.704,Z 384.094,A -85,B 0,C 180,E1 -15355.339,E2 -15355.339} C_VEL
LIN {X 0,Y 325.854,Z 392.576,A -85,B 0,C 180,E1 -15356.078,E2 -15356.078} C_VEL
LIN {X 0,Y 324.918,Z 401.512,A -85,B 0,C 180,E1 -15357.081,E2 -15357.081} C_VEL
LIN {X 0,Y 323.968,Z 408.708,A -85,B 0,C 180,E1 -15358.072,E2 -15358.072} C_VEL
LIN {X 0,Y 322.908,Z 415.689,A -85,B 0,C 180,E1 -15359.238,E2 -15359.238} C_VEL
LIN {X 0,Y 321.882,Z 421.859,A -85,B 0,C 180,E1 -15360.492,E2 -15360.492} C_VEL
LIN {X 0,Y 320.982,Z 427.56,A -85,B 0,C 180,E1 -15361.917,E2 -15361.917} C_VEL
LIN {X 0,Y 320.223,Z 431.935,A -85,B 0,C 180,E1 -15363.262,E2 -15363.262} C_VEL
LIN {X 0,Y 319.513,Z 435.94,A -85,B 0,C 180,E1 -15364.801,E2 -15364.801} C_VEL
LIN {X 0,Y 318.821,Z 439.512,A -85,B 0,C 180,E1 -15366.623,E2 -15366.623} C_VEL
LIN {X 0,Y 318.444,Z 441.334,A -85,B 0,C 180,E1 -15367.964,E2 -15367.964} C_VEL
LIN {X 0,Y 318.126,Z 442.586,A -85,B 0,C 180,E1 -15369.301,E2 -15369.301} C_VEL
LIN {X 0,Y 317.914,Z 443.301,A -85,B 0,C 180,E1 -15370.634,E2 -15370.634} C_VEL
LIN {X 0,Y 317.823,Z 443.493,A -85,B 0,C 180,E1 -15371.966,E2 -15371.966} C_VEL
LIN {X 0,Y 317.758,Z 443.126,A -85,B 0,C 180,E1 -15373.29,E2 -15373.29} C_VEL
LIN {X 0,Y 317.787,Z 442.154,A -85,B 0,C 180,E1 -15374.61,E2 -15374.61} C_VEL
LIN {X 0,Y 317.971,Z 439.884,A -85,B 0,C 180,E1 -15376.51,E2 -15376.51} C_VEL
LIN {X 0,Y 318.283,Z 435.976,A -85,B 0,C 180,E1 -15378.538,E2 -15378.538} C_VEL
LIN {X 0,Y 318.706,Z 430.753,A -85,B 0,C 180,E1 -15380.48,E2 -15380.48} C_VEL
LIN {X 0,Y 319.085,Z 426.333,A -85,B 0,C 180,E1 -15381.77,E2 -15381.77} C_VEL
LIN {X 0,Y 319.545,Z 421.024,A -85,B 0,C 180,E1 -15383.052,E2 -15383.052} C_VEL
LIN {X 0,Y 320.087,Z 414.624,A -85,B 0,C 180,E1 -15384.33,E2 -15384.33} C_VEL
LIN {X 0,Y 320.785,Z 405.807,A -85,B 0,C 180,E1 -15385.76,E2 -15385.76} C_VEL
LIN {X 0,Y 321.601,Z 395.516,A -85,B 0,C 180,E1 -15387.025,E2 -15387.025} C_VEL
LIN {X 0,Y 322.164,Z 387.377,A -85,B 0,C 180,E1 -15387.812,E2 -15387.812} C_VEL
LIN {X 0,Y 322.601,Z 378.035,A -85,B 0,C 180,E1 -15388.518,E2 -15388.518} C_VEL
LIN {X 0,Y 322.997,Z 368.311,A -85,B 0,C 180,E1 -15389.054,E2 -15389.054} C_VEL
LIN {X 0,Y 323.232,Z 358.951,A -85,B 0,C 180,E1 -15389.397,E2 -15389.397} C_VEL
LIN {X 0,Y 324.013,Z 305.448,A -85,B 0,C 180,E1 -15390.603,E2 -15390.603} C_VEL
LIN {X 0,Y 320.475,Z 284.077,A -85,B 0,C 180,E1 -15391.257,E2 -15391.257} C_VEL
LIN {X 0,Y 319.956,Z 280.442,A -85,B 0,C 180,E1 -15392.518,E2 -15392.518} C_VEL
LIN {X 0,Y 319.909,Z 280.445,A -85,B 0,C 180,E1 -15396.307,E2 -15396.307} C_VEL
LIN {X 0,Y 319.804,Z 280.46,A -85,B 0,C 180,E1 -15398.849,E2 -15398.849} C_VEL
LIN {X 0,Y 319.646,Z 280.478,A -85,B 0,C 180,E1 -15402.702,E2 -15402.702} C_VEL
LIN {X 0,Y 319.649,Z 280.483,A -85,B 0,C 180,E1 -15405.298,E2 -15405.298} C_VEL
LIN {X 0,Y 319.644,Z 280.483,A -85,B 0,C 180,E1 -15409.257,E2 -15409.257} C_VEL
LIN {X 0,Y 319.531,Z 280.497,A -85,B 0,C 180,E1 -15413.323,E2 -15413.323} C_VEL
LIN {X 0,Y 319.541,Z 280.492,A -85,B 0,C 180,E1 -15416.097,E2 -15416.097} C_VEL
LIN {X 0,Y 319.514,Z 280.495,A -85,B 0,C 180,E1 -15418.941,E2 -15418.941} C_VEL
LIN {X 0,Y 319.496,Z 280.498,A -85,B 0,C 180,E1 -15421.866,E2 -15421.866} C_VEL
LIN {X 0,Y 319.553,Z 280.495,A -85,B 0,C 180,E1 -15425.546,E2 -15425.546} C_VEL
LIN {X 0,Y 319.504,Z 280.501,A -85,B 0,C 180,E1 -15429.666,E2 -15429.666} C_VEL
LIN {X 0,Y 319.498,Z 280.499,A -85,B 0,C 180,E1 -15433.464,E2 -15433.464} C_VEL
LIN {X 0,Y 319.534,Z 280.492,A -85,B 0,C 180,E1 -15437.021,E2 -15437.021} C_VEL
LIN {X 0,Y 319.504,Z 280.493,A -85,B 0,C 180,E1 -15439.836,E2 -15439.836} C_VEL
LIN {X 0,Y 318.874,Z 280.574,A -85,B 0,C 180,E1 -15440.888,E2 -15440.888} C_VEL
LIN {X 0,Y 316.017,Z 280.93,A -85,B 0,C 180,E1 -15442.6,E2 -15442.6} C_VEL
LIN {X 0,Y 313.581,Z 281.238,A -85,B 0,C 180,E1 -15443.987,E2 -15443.987} C_VEL
LIN {X 0,Y 312.55,Z 281.362,A -85,B 0,C 180,E1 -15445.062,E2 -15445.062} C_VEL
LIN {X 0,Y 312.476,Z 281.373,A -85,B 0,C 180,E1 -15445.426,E2 -15445.426} C_VEL
LIN {X 0,Y 312.493,Z 281.368,A -85,B 0,C 180,E1 -15448.857,E2 -15448.857} C_VEL
LIN {X 0,Y 312.517,Z 281.37,A -85,B 0,C 180,E1 -15451.825,E2 -15451.825} C_VEL
LIN {X 0,Y 312.537,Z 281.363,A -85,B 0,C 180,E1 -15454.712,E2 -15454.712} C_VEL
LIN {X 0,Y 312.531,Z 281.361,A -85,B 0,C 180,E1 -15458.917,E2 -15458.917} C_VEL
LIN {X 0,Y 312.725,Z 281.414,A -85,B 0,C 180,E1 -15462.597,E2 -15462.597} C_VEL
LIN {X 0,Y 312.721,Z 282.906,A -85,B 0,C 180,E1 -15462.997,E2 -15462.997} C_VEL
LIN {X 0,Y 314.905,Z 301.54,A -85,B 0,C 180,E1 -15463.673,E2 -15463.673} C_VEL
LIN {X 0,Y 315.264,Z 306.233,A -85,B 0,C 180,E1 -15463.837,E2 -15463.837} C_VEL
LIN {X 0,Y 313.98,Z 362.752,A -85,B 0,C 180,E1 -15465.751,E2 -15465.751} C_VEL
LIN {X 0,Y 313.688,Z 373.404,A -85,B 0,C 180,E1 -15466.316,E2 -15466.316} C_VEL
LIN {X 0,Y 313.267,Z 385.402,A -85,B 0,C 180,E1 -15467.205,E2 -15467.205} C_VEL
LIN {X 0,Y 312.886,Z 395.106,A -85,B 0,C 180,E1 -15468.177,E2 -15468.177} C_VEL
LIN {X 0,Y 312.293,Z 404.169,A -85,B 0,C 180,E1 -15469.305,E2 -15469.305} C_VEL
LIN {X 0,Y 311.912,Z 412.669,A -85,B 0,C 180,E1 -15470.603,E2 -15470.603} C_VEL
LIN {X 0,Y 311.545,Z 421.014,A -85,B 0,C 180,E1 -15472.226,E2 -15472.226} C_VEL
LIN {X 0,Y 311.159,Z 427.48,A -85,B 0,C 180,E1 -15473.789,E2 -15473.789} C_VEL
LIN {X 0,Y 311.075,Z 433.053,A -85,B 0,C 180,E1 -15475.469,E2 -15475.469} C_VEL
LIN {X 0,Y 310.833,Z 437.85,A -85,B 0,C 180,E1 -15477.412,E2 -15477.412} C_VEL
LIN {X 0,Y 310.764,Z 440.284,A -85,B 0,C 180,E1 -15478.708,E2 -15478.708} C_VEL
LIN {X 0,Y 310.787,Z 442.09,A -85,B 0,C 180,E1 -15480.004,E2 -15480.004} C_VEL
LIN {X 0,Y 310.879,Z 443.295,A -85,B 0,C 180,E1 -15481.3,E2 -15481.3} C_VEL
LIN {X 0,Y 311.081,Z 443.971,A -85,B 0,C 180,E1 -15482.594,E2 -15482.594} C_VEL
LIN {X 0,Y 311.432,Z 444.125,A -85,B 0,C 180,E1 -15483.886,E2 -15483.886} C_VEL
LIN {X 0,Y 311.838,Z 443.761,A -85,B 0,C 180,E1 -15485.176,E2 -15485.176} C_VEL
LIN {X 0,Y 312.174,Z 442.864,A -85,B 0,C 180,E1 -15486.467,E2 -15486.467} C_VEL
LIN {X 0,Y 312.798,Z 440.584,A -85,B 0,C 180,E1 -15488.301,E2 -15488.301} C_VEL
LIN {X 0,Y 313.671,Z 438.155,A -85,B 0,C 180,E1 -15489.649,E2 -15489.649} C_VEL
LIN {X 0,Y 314.54,Z 435.13,A -85,B 0,C 180,E1 -15490.952,E2 -15490.952} C_VEL
LIN {X 0,Y 316.024,Z 429.275,A -85,B 0,C 180,E1 -15492.853,E2 -15492.853} C_VEL
LIN {X 0,Y 317.543,Z 423.043,A -85,B 0,C 180,E1 -15494.421,E2 -15494.421} C_VEL
LIN {X 0,Y 319.263,Z 415.379,A -85,B 0,C 180,E1 -15495.975,E2 -15495.975} C_VEL
LIN {X 0,Y 320.955,Z 406.549,A -85,B 0,C 180,E1 -15497.362,E2 -15497.362} C_VEL
LIN {X 0,Y 322.388,Z 398.11,A -85,B 0,C 180,E1 -15498.431,E2 -15498.431} C_VEL
LIN {X 0,Y 323.888,Z 387.633,A -85,B 0,C 180,E1 -15499.492,E2 -15499.492} C_VEL
LIN {X 0,Y 325.269,Z 375.465,A -85,B 0,C 180,E1 -15500.393,E2 -15500.393} C_VEL
LIN {X 0,Y 326.364,Z 363.52,A -85,B 0,C 180,E1 -15501.023,E2 -15501.023} C_VEL
LIN {X 0,Y 329.878,Z 315.784,A -85,B 0,C 180,E1 -15502.815,E2 -15502.815} C_VEL
LIN {X 0,Y 325.872,Z 306.922,A -85,B 0,C 180,E1 -15503.93,E2 -15503.93} C_VEL
LIN {X 0,Y 320.669,Z 297.211,A -85,B 0,C 180,E1 -15505.416,E2 -15505.416} C_VEL
LIN {X 0,Y 317.061,Z 291.702,A -85,B 0,C 180,E1 -15506.474,E2 -15506.474} C_VEL
LIN {X 0,Y 314.791,Z 287.973,A -85,B 0,C 180,E1 -15507.242,E2 -15507.242} C_VEL
LIN {X 0,Y 312.542,Z 281.367,A -85,B 0,C 180,E1 -15510.491,E2 -15510.491} C_VEL
LIN {X 0,Y 312.516,Z 281.37,A -85,B 0,C 180,E1 -15514.212,E2 -15514.212} C_VEL
LIN {X 0,Y 312.52,Z 281.37,A -85,B 0,C 180,E1 -15517.389,E2 -15517.389} C_VEL
LIN {X 0,Y 312.451,Z 281.377,A -85,B 0,C 180,E1 -15520.719,E2 -15520.719} C_VEL
LIN {X 0,Y 312.462,Z 281.375,A -85,B 0,C 180,E1 -15524.212,E2 -15524.212} C_VEL
LIN {X 0,Y 312.494,Z 281.37,A -85,B 0,C 180,E1 -15527.921,E2 -15527.921} C_VEL
LIN {X 0,Y 312.506,Z 281.371,A -85,B 0,C 180,E1 -15530.972,E2 -15530.972} C_VEL
LIN {X 0,Y 312.541,Z 281.362,A -85,B 0,C 180,E1 -15534.221,E2 -15534.221} C_VEL
LIN {X 0,Y 312.515,Z 281.371,A -85,B 0,C 180,E1 -15537.335,E2 -15537.335} C_VEL
LIN {X 0,Y 312.543,Z 281.451,A -85,B 0,C 180,E1 -15538.997,E2 -15538.997} C_VEL
LIN {X 0,Y 313.742,Z 284.46,A -85,B 0,C 180,E1 -15539.991,E2 -15539.991} C_VEL
LIN {X 0,Y 314.833,Z 285.924,A -85,B 0,C 180,E1 -15540.586,E2 -15540.586} C_VEL
LIN {X 0,Y 315.898,Z 288.356,A -85,B 0,C 180,E1 -15541.296,E2 -15541.296} C_VEL
LIN {X 0,Y 317.224,Z 290.505,A -85,B 0,C 180,E1 -15541.987,E2 -15541.987} C_VEL
LIN {X 0,Y 318.973,Z 296.302,A -85,B 0,C 180,E1 -15543.254,E2 -15543.254} C_VEL
LIN {X 0,Y 319.699,Z 299.901,A -85,B 0,C 180,E1 -15543.867,E2 -15543.867} C_VEL
LIN {X 0,Y 321.236,Z 304.187,A -85,B 0,C 180,E1 -15544.414,E2 -15544.414} C_VEL
LIN {X 0,Y 324.014,Z 317.828,A -85,B 0,C 180,E1 -15545.662,E2 -15545.662} C_VEL
LIN {X 0,Y 326.176,Z 334.054,A -85,B 0,C 180,E1 -15546.871,E2 -15546.871} C_VEL
LIN {X 0,Y 327.351,Z 347.284,A -85,B 0,C 180,E1 -15547.702,E2 -15547.702} C_VEL
LIN {X 0,Y 327.305,Z 354.447,A -85,B 0,C 180,E1 -15548.049,E2 -15548.049} C_VEL
LIN {X 0,Y 324.529,Z 391.845,A -85,B 0,C 180,E1 -15549.484,E2 -15549.484} C_VEL
LIN {X 0,Y 323.106,Z 403.14,A -85,B 0,C 180,E1 -15550.131,E2 -15550.131} C_VEL
LIN {X 0,Y 321.651,Z 412.696,A -85,B 0,C 180,E1 -15550.868,E2 -15550.868} C_VEL
LIN {X 0,Y 319.879,Z 423.244,A -85,B 0,C 180,E1 -15551.92,E2 -15551.92} C_VEL
LIN {X 0,Y 317.843,Z 433.698,A -85,B 0,C 180,E1 -15553.294,E2 -15553.294} C_VEL
LIN {X 0,Y 316.333,Z 441.238,A -85,B 0,C 180,E1 -15554.537,E2 -15554.537} C_VEL
LIN {X 0,Y 314.759,Z 448.964,A -85,B 0,C 180,E1 -15556.112,E2 -15556.112} C_VEL
LIN {X 0,Y 313.429,Z 455.087,A -85,B 0,C 180,E1 -15557.7,E2 -15557.7} C_VEL
LIN {X 0,Y 312.651,Z 459.126,A -85,B 0,C 180,E1 -15558.985,E2 -15558.985} C_VEL
LIN {X 0,Y 311.684,Z 463.799,A -85,B 0,C 180,E1 -15560.918,E2 -15560.918} C_VEL
LIN {X 0,Y 311.234,Z 466.205,A -85,B 0,C 180,E1 -15562.213,E2 -15562.213} C_VEL
LIN {X 0,Y 310.846,Z 468.654,A -85,B 0,C 180,E1 -15564.18,E2 -15564.18} C_VEL
LIN {X 0,Y 310.794,Z 469.876,A -85,B 0,C 180,E1 -15566.11,E2 -15566.11} C_VEL
LIN {X 0,Y 310.78,Z 470.037,A -85,B 0,C 180,E1 -15567.407,E2 -15567.407} C_VEL
LIN {X 0,Y 310.824,Z 471.257,A -85,B 0,C 180,E1 -15568.704,E2 -15568.704} C_VEL
LIN {X 0,Y 310.86,Z 472.072,A -85,B 0,C 180,E1 -15570,E2 -15570} C_VEL
LIN {X 0,Y 310.763,Z 472.356,A -85,B 0,C 180,E1 -15571.296,E2 -15571.296} C_VEL
LIN {X 0,Y 310.746,Z 472.061,A -85,B 0,C 180,E1 -15572.592,E2 -15572.592} C_VEL
LIN {X 0,Y 310.781,Z 471.302,A -85,B 0,C 180,E1 -15573.89,E2 -15573.89} C_VEL
LIN {X 0,Y 310.832,Z 469.299,A -85,B 0,C 180,E1 -15575.795,E2 -15575.795} C_VEL
LIN {X 0,Y 311.193,Z 466.018,A -85,B 0,C 180,E1 -15577.788,E2 -15577.788} C_VEL
LIN {X 0,Y 311.822,Z 461.401,A -85,B 0,C 180,E1 -15579.732,E2 -15579.732} C_VEL
LIN {X 0,Y 312.606,Z 456.354,A -85,B 0,C 180,E1 -15581.345,E2 -15581.345} C_VEL
LIN {X 0,Y 313.435,Z 451.461,A -85,B 0,C 180,E1 -15582.628,E2 -15582.628} C_VEL
LIN {X 0,Y 314.349,Z 445.585,A -85,B 0,C 180,E1 -15583.906,E2 -15583.906} C_VEL
LIN {X 0,Y 315.527,Z 438.449,A -85,B 0,C 180,E1 -15585.172,E2 -15585.172} C_VEL
LIN {X 0,Y 316.696,Z 430.861,A -85,B 0,C 180,E1 -15586.27,E2 -15586.27} C_VEL
LIN {X 0,Y 317.83,Z 422.926,A -85,B 0,C 180,E1 -15587.203,E2 -15587.203} C_VEL
LIN {X 0,Y 318.771,Z 414.768,A -85,B 0,C 180,E1 -15587.978,E2 -15587.978} C_VEL
LIN {X 0,Y 319.598,Z 406.535,A -85,B 0,C 180,E1 -15588.594,E2 -15588.594} C_VEL
LIN {X 0,Y 320.439,Z 397.664,A -85,B 0,C 180,E1 -15589.082,E2 -15589.082} C_VEL
LIN {X 0,Y 320.987,Z 388.554,A -85,B 0,C 180,E1 -15589.432,E2 -15589.432} C_VEL
LIN {X 0,Y 321.755,Z 348.335,A -85,B 0,C 180,E1 -15590.391,E2 -15590.391} C_VEL
LIN {X 0,Y 318.798,Z 328.898,A -85,B 0,C 180,E1 -15591.119,E2 -15591.119} C_VEL
LIN {X 0,Y 315.087,Z 310.615,A -85,B 0,C 180,E1 -15591.932,E2 -15591.932} C_VEL
LIN {X 0,Y 316.328,Z 300.25,A -85,B 0,C 180,E1 -15594.969,E2 -15594.969} C_VEL
LIN {X 0,Y 314.745,Z 291.1,A -85,B 0,C 180,E1 -15597.964,E2 -15597.964} C_VEL
LIN {X 0,Y 312.497,Z 281.37,A -85,B 0,C 180,E1 -15601.397,E2 -15601.397} C_VEL
LIN {X 0,Y 312.515,Z 281.372,A -85,B 0,C 180,E1 -15604.209,E2 -15604.209} C_VEL
LIN {X 0,Y 312.524,Z 281.368,A -85,B 0,C 180,E1 -15607.385,E2 -15607.385} C_VEL
LIN {X 0,Y 312.498,Z 281.372,A -85,B 0,C 180,E1 -15610.708,E2 -15610.708} C_VEL
LIN {X 0,Y 312.46,Z 281.371,A -85,B 0,C 180,E1 -15614.208,E2 -15614.208} C_VEL
LIN {X 0,Y 312.464,Z 281.373,A -85,B 0,C 180,E1 -15617.923,E2 -15617.923} C_VEL
LIN {X 0,Y 312.485,Z 281.371,A -85,B 0,C 180,E1 -15621.922,E2 -15621.922} C_VEL
LIN {X 0,Y 312.539,Z 281.359,A -85,B 0,C 180,E1 -15624.218,E2 -15624.218} C_VEL
LIN {X 0,Y 312.509,Z 281.371,A -85,B 0,C 180,E1 -15627.331,E2 -15627.331} C_VEL
LIN {X 0,Y 312.526,Z 281.367,A -85,B 0,C 180,E1 -15631.285,E2 -15631.285} C_VEL
LIN {X 0,Y 312.558,Z 281.359,A -85,B 0,C 180,E1 -15634.705,E2 -15634.705} C_VEL
LIN {X 0,Y 312.57,Z 281.358,A -85,B 0,C 180,E1 -15637.524,E2 -15637.524} C_VEL
LIN {X 0,Y 312.588,Z 281.361,A -85,B 0,C 180,E1 -15641.65,E2 -15641.65} C_VEL
LIN {X 0,Y 312.69,Z 281.343,A -85,B 0,C 180,E1 -15645.682,E2 -15645.682} C_VEL
LIN {X 0,Y 312.702,Z 281.331,A -85,B 0,C 180,E1 -15649.638,E2 -15649.638} C_VEL
LIN {X 0,Y 312.856,Z 281.321,A -85,B 0,C 180,E1 -15652.25,E2 -15652.25} C_VEL
LIN {X 0,Y 312.902,Z 281.311,A -85,B 0,C 180,E1 -15653.548,E2 -15653.548} C_VEL
LIN {X 0,Y 312.985,Z 281.3,A -85,B 0,C 180,E1 -15658.709,E2 -15658.709} C_VEL
LIN {X 0,Y 312.984,Z 281.302,A -85,B 0,C 180,E1 -15661.282,E2 -15661.282} C_VEL
LIN {X 0,Y 312.681,Z 281.344,A -85,B 0,C 180,E1 -15663.862,E2 -15663.862} C_VEL
LIN {X 0,Y 312.846,Z 281.321,A -85,B 0,C 180,E1 -15666.47,E2 -15666.47} C_VEL
LIN {X 0,Y 312.747,Z 281.335,A -85,B 0,C 180,E1 -15669.046,E2 -15669.046} C_VEL
LIN {X 0,Y 312.629,Z 281.354,A -85,B 0,C 180,E1 -15672.987,E2 -15672.987} C_VEL
LIN {X 0,Y 312.631,Z 281.345,A -85,B 0,C 180,E1 -15675.645,E2 -15675.645} C_VEL
LIN {X 0,Y 312.621,Z 281.352,A -85,B 0,C 180,E1 -15679.232,E2 -15679.232} C_VEL
LIN {X 0,Y 312.535,Z 281.366,A -85,B 0,C 180,E1 -15682.785,E2 -15682.785} C_VEL
LIN {X 0,Y 312.59,Z 281.357,A -85,B 0,C 180,E1 -15685.931,E2 -15685.931} C_VEL
LIN {X 0,Y 312.524,Z 281.367,A -85,B 0,C 180,E1 -15689.646,E2 -15689.646} C_VEL
LIN {X 0,Y 312.503,Z 281.37,A -85,B 0,C 180,E1 -15693.684,E2 -15693.684} C_VEL
LIN {X 0,Y 312.521,Z 281.366,A -85,B 0,C 180,E1 -15697.379,E2 -15697.379} C_VEL
LIN {X 0,Y 312.507,Z 281.362,A -85,B 0,C 180,E1 -15700.699,E2 -15700.699} C_VEL
LIN {X 0,Y 312.573,Z 281.356,A -85,B 0,C 180,E1 -15704.18,E2 -15704.18} C_VEL
LIN {X 0,Y 312.532,Z 281.368,A -85,B 0,C 180,E1 -15707.9,E2 -15707.9} C_VEL
LIN {X 0,Y 312.557,Z 281.523,A -85,B 0,C 180,E1 -15709.634,E2 -15709.634} C_VEL
LIN {X 0,Y 313.4,Z 285.28,A -85,B 0,C 180,E1 -15710.97,E2 -15710.97} C_VEL
LIN {X 0,Y 321.125,Z 303.63,A -85,B 0,C 180,E1 -15712.132,E2 -15712.132} C_VEL
LIN {X 0,Y 322.724,Z 310.108,A -85,B 0,C 180,E1 -15712.428,E2 -15712.428} C_VEL
LIN {X 0,Y 321.505,Z 361.554,A -85,B 0,C 180,E1 -15713.629,E2 -15713.629} C_VEL
LIN {X 0,Y 321.086,Z 371.089,A -85,B 0,C 180,E1 -15714.015,E2 -15714.015} C_VEL
LIN {X 0,Y 320.377,Z 381.971,A -85,B 0,C 180,E1 -15714.67,E2 -15714.67} C_VEL
LIN {X 0,Y 319.222,Z 393.327,A -85,B 0,C 180,E1 -15715.656,E2 -15715.656} C_VEL
LIN {X 0,Y 318.385,Z 400.87,A -85,B 0,C 180,E1 -15716.506,E2 -15716.506} C_VEL
LIN {X 0,Y 317.453,Z 408.013,A -85,B 0,C 180,E1 -15717.484,E2 -15717.484} C_VEL
LIN {X 0,Y 316.403,Z 414.445,A -85,B 0,C 180,E1 -15718.535,E2 -15718.535} C_VEL
LIN {X 0,Y 315.269,Z 421.235,A -85,B 0,C 180,E1 -15719.897,E2 -15719.897} C_VEL
LIN {X 0,Y 314.293,Z 426.8,A -85,B 0,C 180,E1 -15721.265,E2 -15721.265} C_VEL
LIN {X 0,Y 313.474,Z 431.377,A -85,B 0,C 180,E1 -15722.639,E2 -15722.639} C_VEL
LIN {X 0,Y 312.776,Z 435.048,A -85,B 0,C 180,E1 -15723.986,E2 -15723.986} C_VEL
LIN {X 0,Y 311.909,Z 439.309,A -85,B 0,C 180,E1 -15726.073,E2 -15726.073} C_VEL
LIN {X 0,Y 311.453,Z 441.573,A -85,B 0,C 180,E1 -15727.678,E2 -15727.678} C_VEL
LIN {X 0,Y 311.141,Z 442.698,A -85,B 0,C 180,E1 -15728.814,E2 -15728.814} C_VEL
LIN {X 0,Y 310.908,Z 443.562,A -85,B 0,C 180,E1 -15730.18,E2 -15730.18} C_VEL
LIN {X 0,Y 310.734,Z 443.842,A -85,B 0,C 180,E1 -15731.773,E2 -15731.773} C_VEL
LIN {X 0,Y 310.677,Z 443.545,A -85,B 0,C 180,E1 -15732.898,E2 -15732.898} C_VEL
LIN {X 0,Y 310.682,Z 442.71,A -85,B 0,C 180,E1 -15734.249,E2 -15734.249} C_VEL
LIN {X 0,Y 310.864,Z 440.316,A -85,B 0,C 180,E1 -15736.418,E2 -15736.418} C_VEL
LIN {X 0,Y 311.173,Z 436.992,A -85,B 0,C 180,E1 -15738.272,E2 -15738.272} C_VEL
LIN {X 0,Y 311.404,Z 433.86,A -85,B 0,C 180,E1 -15739.598,E2 -15739.598} C_VEL
LIN {X 0,Y 311.967,Z 427.716,A -85,B 0,C 180,E1 -15741.581,E2 -15741.581} C_VEL
LIN {X 0,Y 312.322,Z 422.583,A -85,B 0,C 180,E1 -15742.906,E2 -15742.906} C_VEL
LIN {X 0,Y 312.9,Z 416.492,A -85,B 0,C 180,E1 -15744.199,E2 -15744.199} C_VEL
LIN {X 0,Y 313.526,Z 409.011,A -85,B 0,C 180,E1 -15745.5,E2 -15745.5} C_VEL
LIN {X 0,Y 314.24,Z 400.969,A -85,B 0,C 180,E1 -15746.635,E2 -15746.635} C_VEL
LIN {X 0,Y 315,Z 390.923,A -85,B 0,C 180,E1 -15747.763,E2 -15747.763} C_VEL
LIN {X 0,Y 315.589,Z 380.232,A -85,B 0,C 180,E1 -15748.644,E2 -15748.644} C_VEL
LIN {X 0,Y 316.032,Z 370.131,A -85,B 0,C 180,E1 -15749.243,E2 -15749.243} C_VEL
LIN {X 0,Y 316.277,Z 360.768,A -85,B 0,C 180,E1 -15749.62,E2 -15749.62} C_VEL
LIN {X 0,Y 317.139,Z 306.263,A -85,B 0,C 180,E1 -15750.886,E2 -15750.886} C_VEL
LIN {X 0,Y 313.403,Z 284.437,A -85,B 0,C 180,E1 -15751.566,E2 -15751.566} C_VEL
LIN {X 0,Y 312.892,Z 281.324,A -85,B 0,C 180,E1 -15752.656,E2 -15752.656} C_VEL
LIN {X 0,Y 312.866,Z 281.323,A -85,B 0,C 180,E1 -15756.449,E2 -15756.449} C_VEL
LIN {X 0,Y 312.734,Z 281.343,A -85,B 0,C 180,E1 -15759.051,E2 -15759.051} C_VEL
LIN {X 0,Y 312.6,Z 281.358,A -85,B 0,C 180,E1 -15762.993,E2 -15762.993} C_VEL
LIN {X 0,Y 312.595,Z 281.358,A -85,B 0,C 180,E1 -15765.652,E2 -15765.652} C_VEL
LIN {X 0,Y 312.599,Z 281.36,A -85,B 0,C 180,E1 -15769.238,E2 -15769.238} C_VEL
LIN {X 0,Y 312.509,Z 281.368,A -85,B 0,C 180,E1 -15772.789,E2 -15772.789} C_VEL
LIN {X 0,Y 312.5,Z 281.37,A -85,B 0,C 180,E1 -15775.911,E2 -15775.911} C_VEL
LIN {X 0,Y 312.467,Z 281.375,A -85,B 0,C 180,E1 -15779.658,E2 -15779.658} C_VEL
LIN {X 0,Y 312.493,Z 281.373,A -85,B 0,C 180,E1 -15783.692,E2 -15783.692} C_VEL
LIN {X 0,Y 312.485,Z 281.373,A -85,B 0,C 180,E1 -15787.391,E2 -15787.391} C_VEL
LIN {X 0,Y 312.417,Z 281.378,A -85,B 0,C 180,E1 -15790.721,E2 -15790.721} C_VEL
LIN {X 0,Y 312.43,Z 281.378,A -85,B 0,C 180,E1 -15794.214,E2 -15794.214} C_VEL
LIN {X 0,Y 312.465,Z 281.376,A -85,B 0,C 180,E1 -15797.923,E2 -15797.923} C_VEL
LIN {X 0,Y 312.517,Z 281.371,A -85,B 0,C 180,E1 -15801.915,E2 -15801.915} C_VEL
LIN {X 0,Y 312.476,Z 281.373,A -85,B 0,C 180,E1 -15805.426,E2 -15805.426} C_VEL
LIN {X 0,Y 311.848,Z 281.457,A -85,B 0,C 180,E1 -15806.501,E2 -15806.501} C_VEL
LIN {X 0,Y 309.054,Z 281.81,A -85,B 0,C 180,E1 -15808.252,E2 -15808.252} C_VEL
LIN {X 0,Y 306.642,Z 282.107,A -85,B 0,C 180,E1 -15809.672,E2 -15809.672} C_VEL
LIN {X 0,Y 305.568,Z 282.234,A -85,B 0,C 180,E1 -15810.77,E2 -15810.77} C_VEL
LIN {X 0,Y 305.461,Z 282.245,A -85,B 0,C 180,E1 -15811.143,E2 -15811.143} C_VEL
LIN {X 0,Y 305.49,Z 282.245,A -85,B 0,C 180,E1 -15814.086,E2 -15814.086} C_VEL
LIN {X 0,Y 305.483,Z 282.24,A -85,B 0,C 180,E1 -15816.982,E2 -15816.982} C_VEL
LIN {X 0,Y 305.661,Z 282.201,A -85,B 0,C 180,E1 -15821.922,E2 -15821.922} C_VEL
LIN {X 0,Y 305.691,Z 282.279,A -85,B 0,C 180,E1 -15822.615,E2 -15822.615} C_VEL
LIN {X 0,Y 305.672,Z 283.055,A -85,B 0,C 180,E1 -15822.833,E2 -15822.833} C_VEL
LIN {X 0,Y 307.351,Z 298.779,A -85,B 0,C 180,E1 -15823.44,E2 -15823.44} C_VEL
